(******************提示*******************)
bAnHaveLightWarn :=FALSE;
bCaHaveLightWarn :=FALSE;
FOR K1:=1 TO 50 DO 
      bAnHaveLightWarn:=bAnHaveLightWarn OR AnAlarm.arrLightWarn[K1];
	  bCaHaveLightWarn:=bCaHaveLightWarn OR CaAlarm.arrLightWarn[K1];
END_FOR
(***DDR负数报警***)
(***DDR负数报警***)
IF arrAxisCtrl[NameNo.CaAxisNo.DriverDDR].Status.fActPos<-1 THEN
	CaAlarm.arrFlowAlarm[30]:=TRUE;
END_IF
IF arrAxisCtrl[NameNo.AnAxisNo.DriverDDR].Status.fActPos<-1 THEN
	AnAlarm.arrFlowAlarm[30]:=TRUE;
END_IF

 IF   stSysState.bReset AND  AnAlarm.arrFlowAlarm[30] THEN
	    arrAxisCtrl[NameNo.AnAxisNo.DriverDDR].Cmd.fSetPos:=360;
		arrAxisCtrl[NameNo.AnAxisNo.DriverDDR].Cmd.bSetPos:=TRUE;
		AnAlarm.arrFlowAlarm[30]:=FALSE;
ELSIF  stSysState.bReset AND CaAlarm.arrFlowAlarm[30] THEN
	    arrAxisCtrl[NameNo.CaAxisNo.DriverDDR].Cmd.fSetPos:=360;
		arrAxisCtrl[NameNo.CaAxisNo.DriverDDR].Cmd.bSetPos:=TRUE;
		CaAlarm.arrFlowAlarm[30]:=FALSE;
 END_IF

 (******************报警复位*****************)
 FOR K3:=1 TO 98 DO 
	IF   stSysState.bReset AND  aAlarm[K3]AND NOT aAlarm[52] AND NOT aAlarm[53] AND NOT aAlarm[54]  THEN
			aAlarm[K3]:=FALSE;
	END_IF
END_FOR

(***气压不足报警***)
IF aAirAlarm_TON.Q THEN
	aAlarm[1]:=TRUE;
END_IF
YL_Q[1]:=aAlarm[1];//气压报警传给叠台；
(*
(*** R角废料清洁提示***)
IF  YL_GVL2[1]>=YL_GVL2[2] THEN//正极R角清废料报警；
	aAlarm[2]:=TRUE;
END_IF

IF  YL_GVL2[1]< 0 THEN//正极R角清废料计数错误；
	aAlarm[4]:=TRUE;
END_IF
///////////////////////////
IF    YL_GVL2[3] >=YL_GVL2[4] THEN//负极R角清废料报警；
	aAlarm[3]:=TRUE;
END_IF

IF  YL_GVL2[3] < 0 THEN//负极R角清废料计数错误；
	aAlarm[5]:=TRUE;
END_IF
/////////////////////////////
//复位
IF   stSysState.bReset AND  (aAlarm[2] OR  aAlarm[4] )THEN
		YL_GVL2[1]:=0;
		aAlarm[2]:=FALSE;
		aAlarm[4]:=FALSE;
END_IF

IF   stSysState.bReset AND  (aAlarm[3] OR  aAlarm[5] )THEN
		YL_GVL2[3]:=0;
		aAlarm[3]:=FALSE;
		aAlarm[5]:=FALSE;
END_IF
*)
(*** 除尘风机报警提示***)
aAlarm[6];//风机未启用报警；
IF NOT ProductPar.iModeEN.bFounctionClose[2] THEN
		IF NOT YL_I[1] OR NOT YL_I[3] OR NOT YL_I[5] OR NOT YL_I[7] THEN//2个5.5KW的吸片风机,2个除尘风机；
			aAlarm[6]:=TRUE;//风机未启用报警；
		END_IF
		IF  YL_I[2] OR YL_I[4] OR YL_I[6] OR YL_I[8]  THEN
			aAlarm[7]:=TRUE;// 风机故障报警；
		END_IF
END_IF
FanTon(IN:=NOT aAlarm[6]AND NOT FanTon.Q,PT:=T#1S,Q=>);
IF FanTon.Q THEN
	FanTonS:=FanTonS+1;
END_IF
IF FanTonS>=3600 THEN
	FanTonH:=FanTonH+1;
	FanTonS:=0;
END_IF
IF FanTonH_Set>=FanTonH THEN
	aAlarm[61]:=TRUE;;//风机寿命报警
END_IF



(*** 除尘毛刷气缸没有升起报警***)

IF stSysState.iMode=1 AND NOT 	arrCyCtrl[NameNo.AnCYNo.PoleBrushDustPush_U].Io.DIOFFSwitch THEN
				aAlarm[8]:=TRUE;//	正极上表面毛刷除尘升降气缸位置异常；
END_IF
IF stSysState.iMode=1 AND NOT	arrCyCtrl[NameNo.AnCYNo.PoleWindDustPush_U].Io.DIOFFSwitch THEN
				aAlarm[9]:=TRUE;//	正极上表面风刀除尘升降气缸位置异常;
END_IF
IF stSysState.iMode=1 AND NOT	arrCyCtrl[NameNo.AnCYNo.PoleBrushDustPush_D].Io.DIOFFSwitch THEN
				aAlarm[10]:=TRUE;//	正极下表面毛刷除尘升降气缸位置异常;
END_IF
IF stSysState.iMode=1 AND NOT	arrCyCtrl[NameNo.AnCYNo.PoleWindDustPush_D].Io.DIOFFSwitch THEN
				aAlarm[11]:=TRUE;//	//	正极下表面风刀除尘升降气缸位置异常;
END_IF
////////////////////////
IF stSysState.iMode=1 AND NOT 	arrCyCtrl[NameNo.CaCYNo.PoleBrushDustPush_U].Io.DIOFFSwitch THEN
				aAlarm[12]:=TRUE;//	负极上表面毛刷除尘升降气缸位置异常；
END_IF
IF stSysState.iMode=1 AND NOT	arrCyCtrl[NameNo.CaCYNo.PoleWindDustPush_U].Io.DIOFFSwitch THEN
				aAlarm[13]:=TRUE;//	负极上表面风刀除尘升降气缸位置异常;
END_IF
IF stSysState.iMode=1 AND NOT	arrCyCtrl[NameNo.CaCYNo.PoleBrushDustPush_D].Io.DIOFFSwitch THEN
				aAlarm[14]:=TRUE;//	负极下表面毛刷除尘升降气缸位置异常;
END_IF
IF stSysState.iMode=1 AND NOT	arrCyCtrl[NameNo.CaCYNo.PoleWindDustPush_D].Io.DIOFFSwitch THEN
				aAlarm[15]:=TRUE;//	负极下表面风刀除尘升降气缸位置异常;
END_IF

(*** 安全光栅报警***)
IF NOT AnSenser.biSafetyCurtain_M THEN
	aAlarm[16]:=TRUE;
END_IF
IF NOT AnSenser.biSafetyCurtain_C THEN
	aAlarm[17]:=TRUE;
END_IF		
	
IF NOT CaSenser.biSafetyCurtain_M THEN
	aAlarm[18]:=TRUE;
END_IF
IF NOT CaSenser.biSafetyCurtain_C THEN
	aAlarm[19]:=TRUE;
END_IF	
	
(***************风速仪报警**************)
(***************风速仪报警**************)

aTime[1](IN:=I107[8],PT:=T#20S,Q=>	);
aTime[2](IN:=I107[9],PT:=T#20S,Q=>	);
aTime[3](IN:=I107[10],PT:=T#20S,Q=>	);
aTime[4](IN:=I107[11],PT:=T#20S,Q=>	);
aTime[5](IN:=I107[12],PT:=T#20S,Q=>	);

aTime[6](IN:=I207[8],PT:=T#20S,Q=>	);
aTime[7](IN:=I207[9],PT:=T#20S,Q=>	);
aTime[8](IN:=I207[10],PT:=T#20S,Q=>	);
aTime[9](IN:=I207[11],PT:=T#20S,Q=>	);
aTime[10](IN:=I207[12],PT:=T#20S,Q=>);

IF NOT ProductPar.iModeEN.bFounctionClose[1] THEN//风速仪屏蔽
	IF aTime[1].Q THEN
		aAlarm[20]:=TRUE;
	END_IF
	IF aTime[2].Q THEN
		aAlarm[21]:=TRUE;
	END_IF
	IF aTime[3].Q THEN
		aAlarm[22]:=TRUE;
	END_IF
	IF aTime[4].Q THEN
		aAlarm[23]:=TRUE;
	END_IF
	IF aTime[5].Q THEN
		aAlarm[24]:=TRUE;
	END_IF
	IF aTime[6].Q THEN
		aAlarm[25]:=TRUE;
	END_IF
	IF aTime[7].Q THEN
		aAlarm[26]:=TRUE;
	END_IF
	IF aTime[8].Q THEN
		aAlarm[27]:=TRUE;
	END_IF
	IF aTime[9].Q THEN
		aAlarm[28]:=TRUE;
	END_IF
	IF aTime[10].Q THEN
		aAlarm[29]:=TRUE;
	END_IF
ELSE
	FOR i:=20 TO 29 DO
		aAlarm[i]:=FALSE;
	END_FOR	
END_IF
(******************毛刷感应报警********************)
FOR K4:=30 TO 47 DO 
     aAlarm[48]:=  aAlarm[K4];
END_FOR
(*
(***********摆杆电机扭矩值设置过小报警************)
IF iTargetTorque[1]>-20 THEN
	aAlarm[50]:=TRUE;//正极；
END_IF
IF iTargetTorque[2]>-20 THEN
	aAlarm[51]:=TRUE;//负极；
END_IF
*)
(****************模切清洁报警*********************)

CleanTrig(CLK:= (ProductPar.CleanTimeHMIHour1 = System.StTime.wHour AND ProductPar.CleanTimeHMIMin1 =System.stTime.wMinute)
OR (ProductPar.CleanTimeHMIHour2 = System.StTime.wHour AND ProductPar.CleanTimeHMIMin2 =System.stTime.wMinute)
OR (ProductPar.CleanTimeHMIHour3 = System.StTime.wHour AND ProductPar.CleanTimeHMIMin3 =System.stTime.wMinute)
OR (ProductPar.CleanTimeHMIHour4 = System.StTime.wHour AND ProductPar.CleanTimeHMIMin4 =System.stTime.wMinute));
IF CleanTrig.Q THEN
	aAlarm[52]:=TRUE;//请清洁机台
END_IF
(****************磁棒校验时间报警******************)
AnCibang(CLK:= (ProductPar.CibangTimeHMIHour1 = System.StTime.wHour AND ProductPar.CibangTimeHMIDay1 =System.stTime.wDay));
CaCibang(CLK:= (ProductPar.CibangTimeHMIHour2 = System.StTime.wHour AND ProductPar.CibangTimeHMIDay2 =System.stTime.wDay));
IF AnCibang.Q THEN
	aAlarm[53]:=TRUE;//正极磁棒校验时间报警
END_IF
IF CaCibang.Q THEN
	aAlarm[54]:=TRUE;//负极磁棒校验时间报警
END_IF
(****************模切毛刷清洁时间****************)
AnCleanBrush(CLK:= (ProductPar.BrushTimeHMIHour1 = System.StTime.wHour AND ProductPar.BrushTimeHMIDay1 =System.stTime.wDay));
CaCleanBrush(CLK:= (ProductPar.BrushTimeHMIHour2 = System.StTime.wHour AND ProductPar.BrushTimeHMIDay2 =System.stTime.wDay));
IF AnCleanBrush.Q THEN
	aAlarm[62]:=TRUE;//正极毛刷清洁时间报警
END_IF
IF CaCleanBrush.Q THEN
	aAlarm[63]:=TRUE;//负极毛刷清洁时间报警
END_IF

IF NOT  DTM_Mes1.bFuncEN[0] AND NOT ProductPar.iModeEN.bP2PartEN AND (DTM_Mes1.bFuncEN[1] OR DTM_Mes1.bFuncEN[2] OR DTM_Mes1.bFuncEN[3] OR
	        DTM_Mes1.bFuncEN[4] OR DTM_Mes1.bFuncEN[5] OR DTM_Mes1.bFuncEN[6] OR DTM_Mes1.bFuncEN[7] )  THEN
		 aAlarm[64]:=TRUE;//模切有功能屏蔽报警
END_IF		
			


 AnAlarm.arrFlowAlarm[9];
AnAlarm.arrFlowAlarm[10];
AnAlarm.arrFlowAlarm[11];
AnAlarm.arrFlowAlarm[12];
AnAlarm.arrFlowAlarm[13];
CaAlarm.arrFlowAlarm[9];
CaAlarm.arrFlowAlarm[10];
CaAlarm.arrFlowAlarm[11];
CaAlarm.arrFlowAlarm[12];
CaAlarm.arrFlowAlarm[13];
(*===============================================报警信息============================================================*)
(*****************报警汇总****************)////根据实际情况汇总
//正极报警汇总
arrError[1]:=bAnAxisHaveAlarm OR bAnCYHaveAlarm OR bAnTenHaveAlarm OR bAnCreatTableHaveAlarm OR bAnCamHaveAlarm OR bAnGearHaveAlarm OR bAnFlowHaveAlarm OR aAlarm[16] OR aAlarm[17] OR aAlarm[49]
		OR AnAlarm.arrFlowAlarm[9] OR AnAlarm.arrFlowAlarm[10] OR AnAlarm.arrFlowAlarm[11] OR AnAlarm.arrFlowAlarm[12] OR AnAlarm.arrFlowAlarm[13]
		OR CaAlarm.arrFlowAlarm[9] OR CaAlarm.arrFlowAlarm[10] OR CaAlarm.arrFlowAlarm[11] OR CaAlarm.arrFlowAlarm[12] OR CaAlarm.arrFlowAlarm[13] OR CuterCountAlarm[3];
//负极报警汇总
arrError[2]:=bCaAxisHaveAlarm OR bCaCYHaveAlarm OR bCaTenHaveAlarm OR bCaCreatTableHaveAlarm OR bCaCamHaveAlarm OR bCaGearHaveAlarm OR bCaFlowHaveAlarm OR aAlarm[18] OR aAlarm[19] OR aAlarm[49]
		OR AnAlarm.arrFlowAlarm[9] OR AnAlarm.arrFlowAlarm[10] OR AnAlarm.arrFlowAlarm[11] OR AnAlarm.arrFlowAlarm[12] OR AnAlarm.arrFlowAlarm[13]
		OR CaAlarm.arrFlowAlarm[9] OR CaAlarm.arrFlowAlarm[10] OR CaAlarm.arrFlowAlarm[11] OR CaAlarm.arrFlowAlarm[12] OR CaAlarm.arrFlowAlarm[13] OR CuterCountAlarm[6];
//提示
arrError[3]:=(ProductPar.iModeEN.iModeRun=0 AND (bAnHaveLightWarn OR bCaHaveLightWarn)) OR
				   (ProductPar.iModeEN.iModeRun=1 AND bAnHaveLightWarn) OR 
				   (ProductPar.iModeEN.iModeRun=2 AND bCaHaveLightWarn);

arrError[4];
arrError[5]:=CaAlarm.arrFlowAlarm[30] OR AnAlarm.arrFlowAlarm[30] OR aAlarm[1] OR aAlarm[2] OR aAlarm[3] OR aAlarm[4] OR aAlarm[5]  OR aAlarm[6] OR aAlarm[7] OR aAlarm[8] OR aAlarm[9]
					OR aAlarm[10] OR aAlarm[11] OR aAlarm[12] OR aAlarm[13] OR aAlarm[14] OR aAlarm[15]OR aAlarm[52]OR aAlarm[53]OR aAlarm[54] ;

stSysState.bErrorStop:=(ProductPar.iModeEN.iModeRun=0 AND (arrError[1] OR arrError[2])) OR
								   (ProductPar.iModeEN.iModeRun=1 AND arrError[1]) OR 
								   (ProductPar.iModeEN.iModeRun=2 AND arrError[2])OR arrError[5] OR aAlarm[64];
								   
								   
rDoorAlm[1](CLK:=(AnAlarm.arrFlowAlarm[9] OR AnAlarm.arrFlowAlarm[10] OR AnAlarm.arrFlowAlarm[11] OR AnAlarm.arrFlowAlarm[12] OR AnAlarm.arrFlowAlarm[13]) AND NOT
                            bAnAxisHaveAlarm AND NOT bAnCYHaveAlarm AND NOT bAnTenHaveAlarm AND NOT bAnCreatTableHaveAlarm AND NOT bAnCamHaveAlarm AND NOT
                           bAnGearHaveAlarm AND NOT bAnFlowHaveAlarm AND NOT aAlarm[16] AND NOT aAlarm[17] AND NOT aAlarm[49]  AND NOT CuterCountAlarm[3] );
rDoorAlm[2](CLK:=(CaAlarm.arrFlowAlarm[9] OR CaAlarm.arrFlowAlarm[10] OR CaAlarm.arrFlowAlarm[11] OR CaAlarm.arrFlowAlarm[12] OR CaAlarm.arrFlowAlarm[13]) AND NOT 
                            bCaAxisHaveAlarm AND NOT bCaCYHaveAlarm AND NOT bCaTenHaveAlarm AND NOT bCaCreatTableHaveAlarm AND NOT bCaCamHaveAlarm AND NOT 
                            bCaGearHaveAlarm AND NOT bCaFlowHaveAlarm AND NOT aAlarm[18] AND NOT aAlarm[19] AND NOT aAlarm[49]AND NOT CuterCountAlarm[6] );
IF 	rDoorAlm[1].Q OR bCaDoorALM THEN						
	bAnDoorALM:=TRUE;
END_IF			

IF 	rDoorAlm[1].Q THEN						
	bCaDoorALM:=TRUE;
END_IF		

IF NOT stSysState.bErrorStop AND bAnDoorALM THEN
	bAnDoorALM:=FALSE;
END_IF		
	
IF NOT stSysState.bErrorStop AND bCaDoorALM THEN
	bCaDoorALM:=FALSE;
END_IF				
(*==============报警复位=========================*)
//轴  气缸报警  红灯亮       蜂鸣器 0.5秒 频率 响 8 秒后停止    

IF stSysState.iMode=3 THEN
	stSysState.bReset:=stSysState.btnReset;
END_IF

(*****蜂鸣器*****)
rt100(CLK:=stSysState.bErrorStop, Q=> );
rt101(CLK:=arrError[3]  , Q=> );
IF rt100.Q THEN
	iErrorSetp:=100;//故障报警
END_IF

IF rt101.Q THEN
	iErrorSetp:=200;//警告报警
END_IF


tDelayBuzze(IN:= , PT:= , Q=> , ET=> );
CASE iErrorSetp   OF
100:
  tDelayBuzze.PT:=T#8S;
  tDelayBuzze.IN:=TRUE;
  iErrorSetp:=500;
200:
  tDelayBuzze.PT:=T#4S;
   tDelayBuzze.IN:=TRUE;
  iErrorSetp:=600;
500:
		stSysState.boBuzzer:= Pulse._250ms.Q;  //   (NOT bError1 AND NOT bError2) AND
		IF tDelayBuzze.Q  THEN
			iErrorSetp:=0;
			tDelayBuzze.IN:=FALSE;
			stSysState.boBuzzer:=FALSE;
		END_IF
600:
	IF stSysState.iMode=1 AND NOT stSysState.bErrorStop THEN
		stSysState.boRedLight:=Pulse._1s.Q;
	END_IF
		stSysState.boBuzzer:= Pulse._1s.Q;  //    (NOT bError1 AND NOT bError2) AND
		IF tDelayBuzze.Q  THEN
			iErrorSetp:=0;
			tDelayBuzze.IN:=FALSE;
			IF stSysState.iMode=1 AND NOT stSysState.bErrorStop THEN
				stSysState.boRedLight:=FALSE;
			END_IF
			stSysState.boBuzzer:=FALSE;
		END_IF

END_CASE


(*****三色灯控制*********)
//自动   绿
    RT200[1](CLK:=stSysState.iMode=1 AND NOT stSysState.bErrorStop , Q=> ); 
   IF RT200[1].Q THEN
	  bTurnOn:=TRUE;
      iLightSel:=3;
   END_IF       
//手动  黄
    RT200[2](CLK:=stSysState.iMode=3 AND NOT stSysState.bErrorStop , Q=> ); 
   IF RT200[2].Q THEN
	  bTurnOn:=TRUE;
      iLightSel:=2;
   END_IF 

//暂停   黄
    RT200[3](CLK:=stSysState.iMode=2 AND NOT stSysState.bErrorStop , Q=> ); 
   IF RT200[3].Q THEN
	  bTurnOn:=TRUE;
      iLightSel:=2;
   END_IF 
   
//暂停   红   //急停 OR 故障
    RT200[4](CLK:=stSysState.iMode=4  OR stSysState.bErrorStop  , Q=> ); 
   IF RT200[4].Q THEN
	  bTurnOn:=TRUE;
      iLightSel:=1;
   END_IF    
   
IF bTurnOn THEN
	CASE iLightSel OF 
	  1: //红灯
		stSysState.boGreenLight:=FALSE;
		stSysState.boRedLight:=TRUE;
		stSysState.boYellowLight:=FALSE;
	
	  2://黄灯
		stSysState.boGreenLight:=FALSE;
		stSysState.boRedLight:=FALSE;
		stSysState.boYellowLight:=TRUE;
	
	  3://绿灯
		stSysState.boGreenLight:=TRUE;
		stSysState.boRedLight:=FALSE;
		stSysState.boYellowLight:=FALSE;
	
	END_CASE
   bTurnOn:=FALSE;
END_IF
arrAxis[4].Status.Homed;
arrAxis[5].Status.Homed;
arrAxis[6].Status.Homed;
arrAxis[7].Status.Homed;
arrAxis[8].Status.Homed;
arrAxis[9].Status.Homed;
arrAxis[10].Status.Homed;
arrAxis[11].Status.Homed;
arrAxis[12].Status.Homed;
arrAxis[13].Status.Homed;
arrAxis[14].Status.Homed;
arrAxis[15].Status.Homed;
arrAxis[16].Status.Homed;
arrAxis[17].Status.Homed;
arrAxis[18].Status.Homed;
arrAxis[19].Status.Homed;
arrAxis[20].Status.Homed;
arrAxis[21].Status.Homed;
arrAxis[22].Status.Homed;
arrAxis[23].Status.Homed;
arrAxis[24].Status.Homed;
arrAxis[25].Status.Homed;
arrAxis[26].Status.Homed;
arrAxis[27].Status.Homed;
arrAxis[28].Status.Homed;
arrAxis[29].Status.Homed;
arrAxis[30].Status.Homed;
arrAxis[31].Status.Homed;
arrAxis[32].Status.Homed;
arrAxis[33].Status.Homed;
arrAxis[34].Status.Homed;
arrAxis[35].Status.Homed;
arrAxis[36].Status.Homed;
arrAxis[37].Status.Homed;
arrAxis[38].Status.Homed;
arrAxis[39].Status.Homed;
arrAxis[40].Status.Homed;
arrAxis[41].Status.Homed;
arrAxis[42].Status.Homed;
arrAxis[43].Status.Homed;
arrAxis[44].Status.Homed;
arrAxis[45].Status.Homed;
arrAxis[46].Status.Homed;
arrAxis[47].Status.Homed;
arrAxis[48].Status.Homed;
arrAxis[49].Status.Homed;
arrAxis[50].Status.Homed;
arrAxis[51].Status.Homed;
arrAxis[52].Status.Homed;
arrAxis[53].Status.Homed;
arrAxis[54].Status.Homed;
arrAxis[55].Status.Homed;
arrAxis[56].Status.Homed;
arrAxis[57].Status.Homed;
arrAxis[58].Status.Homed;
arrAxis[59].Status.Homed;
arrAxis[60].Status.Homed;
END_ACTION

ACTION Condition:
//按钮汇总
stSysState.btnAuto:=AnSys.btnAuto AND CaSys.btnAuto ;
stSysState.btnStart:=AnSys.btnStart OR CaSys.btnStart;
stSysState.btnStop:=AnSys.btnStop OR CaSys.btnStop;
stSysState.btnReset:=AnSys.btnReset OR CaSys.btnReset;
bEncloserEstop:=(NOT AnBtn.EncloserEstop[1] OR NOT AnBtn.EncloserEstop[2] OR NOT AnBtn.EncloserEstop[3] OR 
						  NOT CaBtn.EncloserEstop[1] OR NOT CaBtn.EncloserEstop[2] OR NOT CaBtn.EncloserEstop[3])AND test[1] ;
bBoxEstop:=NOT AnBtn.PoleBoxEStop OR NOT AnBtn.NGBoxEStop OR  NOT CaBtn.PoleBoxEStop OR NOT CaBtn.NGBoxEStop ;

stSysState.btnEstop:=(NOT AnSys.btnEstop OR NOT CaSys.btnEstop //面板急停
								OR bEncloserEstop//外罩急停
								(*OR bBoxEstop//按钮盒急停*)
								) ;//常闭
//面板按钮灯控制
bAnReady:=AnSys.bAutoCondition1 AND AnSys.Homed AND NOT AnSys.hmiDisCamAll;
bCaReady:=CaSys.bAutoCondition1 AND CaSys.Homed AND NOT CaSys.hmiDisCamAll;

AnSys.boStartLight:=stSysState.boGreenLight OR bAnReady AND Pulse._500ms.Q OR AnSys.btnStart;
CaSys.boStartLight:=stSysState.boGreenLight OR bCaReady AND Pulse._500ms.Q OR AnSys.btnStart;

AnSys.boStopLight:=AnSys.Stoping AND Pulse._250ms.Q OR AnSys.btnStop;
CaSys.boStopLight:=CaSys.Stoping AND Pulse._250ms.Q OR CaSys.btnStop;

AnSys.boResetLight:=stSysState.boRedLight AND Pulse._500ms.Q OR AnSys.btnReset;
CaSys.boResetLight:=stSysState.boRedLight AND Pulse._500ms.Q OR CaSys.btnReset;		
////////////////////////////////////////////设备状态//////////////////////
	IF stSysState.btnEstop THEN
		stSysState.iModehmi:=4;
	ELSIF NOT stSysState.btnEstop AND stSysState.bErrorStop THEN
		stSysState.iModehmi:=5;
	ELSIF NOT stSysState.btnEstop AND NOT stSysState.bErrorStop AND stSysState.FlgManua AND stSysState.iMode=3THEN
		stSysState.iModehmi:=3;
	ELSIF NOT stSysState.btnEstop AND NOT stSysState.bErrorStop AND ((NOT stSysState.FlgManua AND stSysState.FlgAuto AND stSysState.iMode=1) OR stSysState.iMode=1) THEN
		stSysState.iModehmi:=1;
	ELSIF NOT stSysState.btnEstop AND NOT stSysState.bErrorStop AND NOT stSysState.FlgManua AND stSysState.FlgAuto AND stSysState.iMode<>1 AND
		 	((ProductPar.iModeEN.iModeRun=0 AND bAnReady AND bCaReady) OR (ProductPar.iModeEN.iModeRun=1 AND bAnReady) OR (ProductPar.iModeEN.iModeRun=2 AND bCaReady))
			THEN	
		stSysState.iModehmi:=2;	
	ELSE
		stSysState.iModehmi:=6;	
	END_IF		
	P2Interaction.bP1Runing:=stSysState.iModehmi=1;
////////////////////////////////////////////主流程与分模块交互//////////////////////
(*
stSysState.bAutoCondition:=((AnSys.bAutoCondition1 AND AnSys.Homed AND NOT AnSys.hmiDisCamAll AND 
			CaSys.bAutoCondition1 AND CaSys.Homed AND NOT CaSys.hmiDisCamAll AND
			ProductPar.iModeEN.iModeRun=0) OR//正负同时启用
			(AnSys.bAutoCondition1 AND AnSys.Homed AND NOT AnSys.hmiDisCamAll AND
			ProductPar.iModeEN.iModeRun=1) OR//仅正极启用
			(CaSys.bAutoCondition1 AND CaSys.Homed AND NOT CaSys.hmiDisCamAll AND
			ProductPar.iModeEN.iModeRun=2))//仅负极启用
			AND NOT stSysState.bErrorStop;
*)
stSysState.bAutoCondition:=	(AnSys.bAutoCondition1 AND AnSys.Homed AND NOT AnSys.hmiDisCamAll AND CaSys.bAutoCondition1 AND CaSys.Homed AND NOT CaSys.hmiDisCamAll AND ProductPar.iModeEN.iModeRun=0 
	AND	( (ProductPar.AnPar.MQ.bWindSelect AND  Ansys.PolePieceNumberOK1)  OR ( NOT ProductPar.AnPar.MQ.bWindSelect AND  Ansys.PolePieceNumberOK2) )
	AND  ( ( ProductPar.CaPar.MQ.bWindSelect AND  Casys.PolePieceNumberOK1 ) OR (  NOT ProductPar.CaPar.MQ.bWindSelect AND  Casys.PolePieceNumberOK2 ) ) ) OR //正负同时启用

		(AnSys.bAutoCondition1 AND AnSys.Homed AND NOT AnSys.hmiDisCamAll AND ProductPar.iModeEN.iModeRun=1  AND
		 ( ( ProductPar.AnPar.MQ.bWindSelect AND  Ansys.PolePieceNumberOK1 ) OR (  NOT ProductPar.AnPar.MQ.bWindSelect AND  Ansys.PolePieceNumberOK2 ) )) OR//仅正极启用
	
		(CaSys.bAutoCondition1 AND CaSys.Homed AND NOT CaSys.hmiDisCamAll AND ProductPar.iModeEN.iModeRun=2 AND 
		  ( ( ProductPar.CaPar.MQ.bWindSelect AND  Casys.PolePieceNumberOK1 ) OR (  NOT ProductPar.CaPar.MQ.bWindSelect AND  Casys.PolePieceNumberOK2 )  ) )//仅负极启用
		  AND NOT stSysState.bErrorStop; 			
Ansys.bAutoTen:=stSysState.iMode=1 AND (ProductPar.iModeEN.iModeRun=0 OR ProductPar.iModeEN.iModeRun=1);
Casys.bAutoTen:=stSysState.iMode=1 AND (ProductPar.iModeEN.iModeRun=0 OR ProductPar.iModeEN.iModeRun=2);
Ansys.bAutoMain:=AnSys.bAutoCondition2 AND ((ProductPar.iModeEN.iModeRun=0 AND CaSys.bAutoCondition2) OR ProductPar.iModeEN.iModeRun=1);
Casys.bAutoMain:=CaSys.bAutoCondition2 AND ((ProductPar.iModeEN.iModeRun=0 AND AnSys.bAutoCondition2) OR ProductPar.iModeEN.iModeRun=2);

stSysState.bStopFinished:=(AnSys.bStopFinished AND CaSys.bStopFinished  AND ProductPar.iModeEN.iModeRun=0) OR//正负同时启用
			(AnSys.bStopFinished AND ProductPar.iModeEN.iModeRun=1) OR//仅正极启用
			(CaSys.bStopFinished AND ProductPar.iModeEN.iModeRun=2);//仅负极启用

///////////////////////////////////交互映射/////////////////////////////////////
//////////叠片TO模切//////////
//一号叠台正极
AnInter.M1Done:=D_Pro.bAn_M1Done;
AnInter.M1Safety:=D_Pro.bAn_M1Safety;
AnInter.iM1Ask:=D_Sys.iAn1Ask;
AnInter.M1LockReady:=D_Pro.bAn_M1LockReady;
AnInter.M1JumpReady:=D_Pro.bAn_M1JumpReady;
AnInter.M1PoleHave:=D_Pro.bAn_M1PoleHave;


//一号叠台负极
CaInter.M1Done:=D_Pro.bCa_M1Done;
CaInter.M1Safety:=D_Pro.bCa_M1Safety;
CaInter.iM1Ask:=D_Sys.iCa1Ask;
CaInter.M1LockReady:=D_Pro.bCa_M1LockReady;
CaInter.M1JumpReady:=D_Pro.bCa_M1JumpReady;
CaInter.M1PoleHave:=D_Pro.bCa_M1PoleHave;


//二号叠台正极
AnInter.M2Done:=D_Pro.bAn_M2Done;
AnInter.M2Safety:=D_Pro.bAn_M2Safety;
AnInter.iM2Ask:=D_Sys.iAn2Ask;
AnInter.M2LockReady:=D_Pro.bAn_M2LockReady;
AnInter.M2JumpReady:=D_Pro.bAn_M2JumpReady;
AnInter.M2PoleHave:=D_Pro.bAn_M2PoleHave;


//二号叠台负极
CaInter.M2Done:=D_Pro.bCa_M2Done;
CaInter.M2Safety:=D_Pro.bCa_M2Safety;
CaInter.iM2Ask:=D_Sys.iCa2Ask;
CaInter.M2LockReady:=D_Pro.bCa_M2LockReady;
CaInter.M2JumpReady:=D_Pro.bCa_M2JumpReady;
CaInter.M2PoleHave:=D_Pro.bCa_M2PoleHave;


//三号叠台正极
AnInter.M3Done:=D_Pro.bAn_M3Done;
AnInter.M3Safety:=D_Pro.bAn_M3Safety;
AnInter.iM3Ask:=D_Sys.iAn3Ask;
AnInter.M3LockReady:=D_Pro.bAn_M3LockReady;
AnInter.M3JumpReady:=D_Pro.bAn_M3JumpReady;
AnInter.M3PoleHave:=D_Pro.bAn_M3PoleHave;


//三号叠台负极
CaInter.M3Done:=D_Pro.bCa_M3Done;
CaInter.M3Safety:=D_Pro.bCa_M3Safety;
CaInter.iM3Ask:=D_Sys.iCa3Ask;
CaInter.M3LockReady:=D_Pro.bCa_M3LockReady;
CaInter.M3JumpReady:=D_Pro.bCa_M3JumpReady;
CaInter.M3PoleHave:=D_Pro.bCa_M3PoleHave;


//公共
P2Interaction.bP2ClearDo:=D_Sys.bP2ClearDo;
P2Interaction.bP2ClearDone:=D_Sys.bP2ClearDone;
P2Interaction.P2M1Enable:=D_Sys.bP2M1Enable;//叠台工位：1=屏蔽   模切工位：1=启用，故取反。
P2Interaction.P2M2Enable:=D_Sys.bP2M2Enable;//叠台工位：1=屏蔽   模切工位：1=启用，故取反。
P2Interaction.P2M3Enable:=D_Sys.bP2M3Enable;//叠台工位：1=屏蔽   模切工位：1=启用，故取反。
P2Interaction.bP2Estop:=D_Sys.bP2Estop;
P2Interaction.bP2Runing:=D_Sys.bP2Runing;
P2Interaction.bP2Start:=D_Sys.bP2Start;

///////////模切TO叠片/////////
//一号叠台正极
M_Pro.bAn_M1Allow:=AnInter.M1Allow;
M_Pro.bAn_M1Allow2:=AnInter.M1Allow2;
//一号叠台负极
M_Pro.bCa_M1Allow:=CaInter.M1Allow;
//M_Pro.bCa_M1Allow:=CaInter.M1Allow2;
//二号叠台正极
M_Pro.bAn_M2Allow:=AnInter.M2Allow;
//M_Pro.bAn_M2Allow2:=AnInter.M2Allow2;
//二号叠台负极
M_Pro.bCa_M2Allow:=CaInter.M2Allow;
//M_Pro.bCa_M2Allow:=CaInter.M2Allow2;
//三号叠台正极
M_Pro.bAn_M3Allow:=AnInter.M3Allow;
//M_Pro.bAn_M3Allow2:=AnInter.M3Allow2;
//三号叠台负极
M_Pro.bCa_M3Allow:=CaInter.M3Allow;
//M_Pro.bCa_M3Allow:=CaInter.M3Allow2;

(*20240404
///////////模切TO叠片/////////
//一号叠台正极
M_Pro.bAn_M1Allow:=AnInter.M1Allow;
//一号叠台负极
M_Pro.bCa_M1Allow:=CaInter.M1Allow;
//二号叠台正极
M_Pro.bAn_M2Allow:=AnInter.M2Allow;
//二号叠台负极
M_Pro.bCa_M2Allow:=CaInter.M2Allow;
//三号叠台正极
M_Pro.bAn_M3Allow:=AnInter.M3Allow;
//三号叠台负极
M_Pro.bCa_M3Allow:=CaInter.M3Allow;
20240404*)
//公共
M_Sys.bP1ClearDo:=P2Interaction.bP1ClearDo;
M_Sys.bP1ClearDone:=P2Interaction.bP1ClearDone;
M_Sys.bP1Estop:=P2Interaction.bP1Estop;
M_Sys.bP1Runing:=P2Interaction.bP1Runing;
M_Sys.bP1Start:=P2Interaction.bP1Start;
M_Sys.iCarryPoleMode:=ProductPar.iModeEN.iCarryPoleMode;
M_Sys.p1state:=stSysState.iModehmi;
IF test[2] THEN
	MEMSET(ADR(PoleData.AnIntervalData),0,SIZEOF(PoleData.AnIntervalData)); //  
	test[2]:=FALSE;
END_IF
IF test[3] THEN
	MEMSET(ADR(PoleData.CaIntervalData),0,SIZEOF(PoleData.CaIntervalData)); //  
	test[3]:=FALSE;
END_IF
IF test[4] THEN
	MEMSET(ADR(PoleData.AnTabData),0,SIZEOF(PoleData.AnTabData)); //  
	test[4]:=FALSE;
END_IF
IF test[5] THEN
	MEMSET(ADR(PoleData.CaTabData),0,SIZEOF(PoleData.CaTabData)); //  
	test[5]:=FALSE;
END_IF
//监控
PoleData.	AnBeltData[1].bHavePole;
PoleData.	AnBeltData[2].bHavePole;
PoleData.	AnBeltData[3].bHavePole;
PoleData.	AnBeltData[4].bHavePole;
PoleData.	AnBeltData[5].bHavePole;
PoleData.	AnBeltData[6].bHavePole;
PoleData.	AnBeltData[7].bHavePole;
PoleData.	AnBeltData[8].bHavePole;
PoleData.	AnBeltData[9].bHavePole;
PoleData.	AnBeltData[10].bHavePole;
PoleData.	AnBeltData[11].bHavePole;
PoleData.	AnBeltData[12].bHavePole;
PoleData.	AnBeltData[13].bHavePole;
PoleData.	AnBeltData[14].bHavePole;
PoleData.	AnBeltData[15].bHavePole;
PoleData.	AnBeltData[16].bHavePole;
PoleData.	AnBeltData[17].bHavePole;
PoleData.	AnBeltData[18].bHavePole;
PoleData.	AnBeltData[19].bHavePole;
PoleData.	AnBeltData[20].bHavePole;
PoleData.	AnBeltData[21].bHavePole;
PoleData.	AnBeltData[22].bHavePole;
PoleData.	AnBeltData[23].bHavePole;
PoleData.	AnBeltData[24].bHavePole;
PoleData.	AnBeltData[25].bHavePole;
PoleData.	AnBeltData[26].bHavePole;
PoleData.	AnBeltData[27].bHavePole;
PoleData.	AnBeltData[28].bHavePole;
PoleData.	AnBeltData[29].bHavePole;
PoleData.	AnBeltData[30].bHavePole;				
stSysState.hmiStart;					
bInitReset;
arrAxisCtrl[NameNo.AnVirAxisNo.VirMain].Status.fModuloActPos;
arrAxisCtrl[NameNo.AnVirAxisNo.VirDriver].Status.fActPos;
arrAxisCtrl[NameNo.AnVirAxisNo.VirBelt].Status.fActPos;
arrAxisCtrl[NameNo.AnAxisNo.Mould].Status.fModuloActPos;
arrAxisCtrl[NameNo.AnAxisNo.Cuter].Status.fModuloActPos;
arrAxisCtrl[NameNo.AnAxisNo.DriverDDR].Status.fActPos;
arrAxisCtrl[NameNo.AnAxisNo.CCDPressPush].Status.fModuloActPos;
//arrAxisCtrl[NameNo.AnAxisNo.NGPush2].Status.fModuloActPos;
arrAxisCtrl[NameNo.AnAxisNo.CuterBelt].Status.fActPos;
arrAxisCtrl[NameNo.AnAxisNo.NGPushReverseBelt].Status.fActPos;
arrAxisCtrl[NameNo.AnAxisNo.DedustBelt].Status.fActPos;
arrAxisCtrl[NameNo.AnAxisNo.DedustReverseBelt].Status.fActPos;
arrAxisCtrl[NameNo.AnAxisNo.SubBelt1].Status.fActPos;
arrAxisCtrl[NameNo.AnAxisNo.SubBelt2].Status.fActPos;
arrAxisCtrl[NameNo.AnAxisNo.SubBelt3].Status.fActPos;

arrAxisCtrl[NameNo.AnAxisNo.CuterBeltChange].Status.Homed;
arrAxisCtrl[NameNo.AnAxisNo.CuterBeltChange].cmd.bHome;

PoleData.	CaBeltData[1].bHavePole;
PoleData.	CaBeltData[2].bHavePole;
PoleData.	CaBeltData[3].bHavePole;
PoleData.	CaBeltData[4].bHavePole;
PoleData.	CaBeltData[5].bHavePole;
PoleData.	CaBeltData[6].bHavePole;
PoleData.	CaBeltData[7].bHavePole;
PoleData.	CaBeltData[8].bHavePole;
PoleData.	CaBeltData[9].bHavePole;
PoleData.	CaBeltData[10].bHavePole;
PoleData.	CaBeltData[11].bHavePole;
PoleData.	CaBeltData[12].bHavePole;
PoleData.	CaBeltData[13].bHavePole;
PoleData.	CaBeltData[14].bHavePole;
PoleData.	CaBeltData[15].bHavePole;
PoleData.	CaBeltData[16].bHavePole;
PoleData.	CaBeltData[17].bHavePole;
PoleData.	CaBeltData[18].bHavePole;
PoleData.	CaBeltData[19].bHavePole;
PoleData.	CaBeltData[20].bHavePole;
PoleData.	CaBeltData[21].bHavePole;
PoleData.	CaBeltData[22].bHavePole;
PoleData.	CaBeltData[23].bHavePole;
PoleData.	CaBeltData[24].bHavePole;
PoleData.	CaBeltData[25].bHavePole;
PoleData.	CaBeltData[26].bHavePole;
PoleData.	CaBeltData[27].bHavePole;
PoleData.	CaBeltData[28].bHavePole;
PoleData.	CaBeltData[29].bHavePole;
PoleData.	CaBeltData[30].bHavePole;	




//正极左卷料号OK
IF  (ProductPar.AnPar.MQ.bWindSelect AND arrCyCtrl[NameNo.AnCYNo.Inflation_L].Status.ONState 
 AND DT_To_MQ_MES.Mes_PcToPlc1 AND  LEN(DT_To_MQ_MES.PostiveCode1)>6  )  OR ProductPar.iModeEN.PartNumberOff THEN
	Ansys.PolePieceNumberOK1:=TRUE;
ELSE
	Ansys.PolePieceNumberOK1:=FALSE;
END_IF

//正极右卷料号OK
IF  (NOT ProductPar.AnPar.MQ.bWindSelect AND arrCyCtrl[NameNo.AnCYNo.Inflation_R].Status.ONState
  AND DT_To_MQ_MES.Mes_PcToPlc2 AND LEN(DT_To_MQ_MES.PostiveCode2)>6  )  OR ProductPar.iModeEN.PartNumberOff THEN
	Ansys.PolePieceNumberOK2:=TRUE;
ELSE
	Ansys.PolePieceNumberOK2:=FALSE;
END_IF

//当前使用左卷
IF ProductPar.AnPar.MQ.bWindSelect THEN
	IF Ansys.PolePieceNumberOK1 THEN
		PoleData.AnBeltData[1].Code:=DT_To_MQ_MES.PostiveCode1;
	ELSE
		PoleData.AnBeltData[1].Code:='';//当前卷物料码异常
	END_IF
ELSE//当前使用右卷
	IF Ansys.PolePieceNumberOK2 THEN
		PoleData.AnBeltData[1].Code:=DT_To_MQ_MES.PostiveCode2;
	ELSE
		PoleData.AnBeltData[1].Code:='';//当前卷物料码异常
	END_IF
END_IF

//正极右卷换左卷---正常换卷
Code_MES[1](CLK:=ProductPar.AnPar.MQ.bWindSelect , Q=> );//AND arrCyCtrl[NameNo.AnCYNo.Inflation_L].Status.ONState  AND  stAnUwindTen.bTensionOK 
IF Code_MES[1].Q THEN
	Ansys.PolePieceNumberOK2:=FALSE;//正极右卷料号OK
	MQ_To_DT_MES.Mes_PlcToPc1:=FALSE;//正极左卷换卷请求
	MQ_To_DT_MES.Mes_PlcToPc2:=TRUE;//正极右卷换卷请求触发
END_IF
//正极左卷换右卷---正常换卷
Code_MES[2](CLK:=NOT ProductPar.AnPar.MQ.bWindSelect  , Q=> );//AND arrCyCtrl[NameNo.AnCYNo.Inflation_R].Status.ONState  AND  stAnUwindTen.bTensionOK
IF Code_MES[2].Q THEN
	Ansys.PolePieceNumberOK1:=FALSE;//正极左卷料号OK
	MQ_To_DT_MES.Mes_PlcToPc1:=TRUE;//正极左卷换卷请求触发
	MQ_To_DT_MES.Mes_PlcToPc2:=FALSE;//正极右卷换卷请求
END_IF

//正极气涨轴切换换卷
Code_MES[3](CLK:=arrCyCtrl[NameNo.AnCYNo.Inflation_L].Io.DOStatus1, Q=> );//左卷
Code_MES[4](CLK:=arrCyCtrl[NameNo.AnCYNo.Inflation_R].Io.DOStatus1, Q=> );//右卷
IF Code_MES[3].Q THEN//左卷请求
	Ansys.PolePieceNumberOK1:=FALSE;//正极左卷料号OK
	MQ_To_DT_MES.Mes_PlcToPc1:=TRUE;//正极左卷换卷请求触发
	MQ_To_DT_MES.Mes_PlcToPc2:=FALSE;//正极右卷换卷请求
END_IF
IF Code_MES[4].Q THEN//右卷请求
	Ansys.PolePieceNumberOK2:=FALSE;//正极右卷料号OK
	MQ_To_DT_MES.Mes_PlcToPc1:=FALSE;//正极左卷换卷请求
	MQ_To_DT_MES.Mes_PlcToPc2:=TRUE;//正极右卷换卷请求触发
END_IF



//负极左卷料号OK
IF  (ProductPar.CaPar.MQ.bWindSelect AND arrCyCtrl[NameNo.CaCYNo.Inflation_L].Status.ONState 
 AND DT_To_MQ_MES.Mes_PcToPlc3 AND  LEN(DT_To_MQ_MES.NegativeCode1)>6  )  OR ProductPar.iModeEN.PartNumberOff THEN
	Casys.PolePieceNumberOK1:=TRUE;
ELSE
	Casys.PolePieceNumberOK1:=FALSE;
END_IF

//负极右卷料号OK
IF  (NOT ProductPar.CaPar.MQ.bWindSelect AND arrCyCtrl[NameNo.CaCYNo.Inflation_R].Status.ONState
  AND DT_To_MQ_MES.Mes_PcToPlc4 AND LEN(DT_To_MQ_MES.NegativeCode2)>6  )  OR ProductPar.iModeEN.PartNumberOff THEN
	Casys.PolePieceNumberOK2:=TRUE;
ELSE
	Casys.PolePieceNumberOK2:=FALSE;
END_IF

IF ProductPar.CaPar.MQ.bWindSelect THEN
	IF  Casys.PolePieceNumberOK1 THEN
		PoleData.CaBeltData[1].Code:=DT_To_MQ_MES.NegativeCode1;
	ELSE
		PoleData.CaBeltData[1].Code:='';//当前卷物料码异常
	END_IF
ELSE
	IF  Casys.PolePieceNumberOK2 THEN
		PoleData.CaBeltData[1].Code:=DT_To_MQ_MES.NegativeCode2;
	ELSE
		PoleData.CaBeltData[1].Code:='';//当前卷物料码异常
	END_IF
END_IF

//负极右卷换左卷---正常换卷
Code_MES[5](CLK:=ProductPar.CaPar.MQ.bWindSelect  , Q=> );//AND arrCyCtrl[NameNo.CaCYNo.Inflation_L].Status.ONState  AND  stCaUwindTen.bTensionOK
IF Code_MES[5].Q THEN
	Casys.PolePieceNumberOK2:=FALSE;//负极右卷料号OK
	MQ_To_DT_MES.Mes_PlcToPc3:=FALSE;//负极左卷换卷请求
	MQ_To_DT_MES.Mes_PlcToPc4:=TRUE;//负极右卷换卷请求触发
END_IF
//正极左卷换右卷---正常换卷
Code_MES[6](CLK:=NOT ProductPar.CaPar.MQ.bWindSelect  , Q=> );//AND arrCyCtrl[NameNo.CaCYNo.Inflation_R].Status.ONState  AND  stCaUwindTen.bTensionOK
IF Code_MES[6].Q THEN
	Casys.PolePieceNumberOK1:=FALSE;//负极左卷料号OK
	MQ_To_DT_MES.Mes_PlcToPc3:=TRUE;//负极左卷换卷请求触发
	MQ_To_DT_MES.Mes_PlcToPc4:=FALSE;//负极右卷换卷请求
END_IF


//负极气涨轴切换换卷
Code_MES[7](CLK:=arrCyCtrl[NameNo.CaCYNo.Inflation_L].Io.DOStatus1, Q=> );//左卷
Code_MES[8](CLK:=arrCyCtrl[NameNo.CaCYNo.Inflation_R].Io.DOStatus1, Q=> );//右卷
IF Code_MES[7].Q THEN//左卷请求
	Casys.PolePieceNumberOK1:=FALSE;//负极左卷料号OK
	MQ_To_DT_MES.Mes_PlcToPc3:=TRUE;//负极左卷换卷请求触发
	MQ_To_DT_MES.Mes_PlcToPc4:=FALSE;//负极右卷换卷请求
END_IF
IF Code_MES[8].Q THEN//右卷请求
	Casys.PolePieceNumberOK2:=FALSE;//负极右卷料号OK
	MQ_To_DT_MES.Mes_PlcToPc3:=FALSE;//负极左卷换卷请求
	MQ_To_DT_MES.Mes_PlcToPc4:=TRUE;//负极右卷换卷请求触发
END_IF



//条码校验未完成提示
IF ProductPar.AnPar.MQ.bWindSelect AND  NOT Ansys.PolePieceNumberOK1  AND NOT ProductPar.iModeEN.PartNumberOff THEN
	AnAlarm.arrLightWarn[41]:=TRUE;//正极左卷物料码校验未通过
ELSE
	AnAlarm.arrLightWarn[41]:=FALSE;//正极左卷物料码校验未通过
END_IF
IF NOT ProductPar.AnPar.MQ.bWindSelect AND NOT Ansys.PolePieceNumberOK2  AND NOT ProductPar.iModeEN.PartNumberOff THEN
	AnAlarm.arrLightWarn[42]:=TRUE;//正极右卷物料码校验未通过
ELSE
	AnAlarm.arrLightWarn[42]:=FALSE;//正极右卷物料码校验未通过
END_IF

IF ProductPar.CaPar.MQ.bWindSelect AND  NOT Casys.PolePieceNumberOK1  AND NOT ProductPar.iModeEN.PartNumberOff THEN
	CaAlarm.arrLightWarn[41]:=TRUE;//负极左卷物料码校验未通过
ELSE
	CaAlarm.arrLightWarn[41]:=FALSE;//负极左卷物料码校验未通过
END_IF
IF NOT  ProductPar.CaPar.MQ.bWindSelect AND NOT Casys.PolePieceNumberOK2  AND NOT ProductPar.iModeEN.PartNumberOff THEN
	CaAlarm.arrLightWarn[42]:=TRUE;//负极右卷物料码校验未通过
ELSE
	CaAlarm.arrLightWarn[42]:=FALSE;//负极右卷物料码校验未通过
END_IF


//触发信号清除
tCode_MES[1](IN:=MQ_To_DT_MES.Mes_PlcToPc1 , PT:=T#0.2S , Q=> , ET=> );
tCode_MES[2](IN:=MQ_To_DT_MES.Mes_PlcToPc2 , PT:=T#0.2S , Q=> , ET=> );
tCode_MES[3](IN:=MQ_To_DT_MES.Mes_PlcToPc3 , PT:=T#0.2S , Q=> , ET=> );
tCode_MES[4](IN:=MQ_To_DT_MES.Mes_PlcToPc4 , PT:=T#0.2S , Q=> , ET=> );
IF tCode_MES[1].Q THEN
	MQ_To_DT_MES.Mes_PlcToPc1:=FALSE;//正极左卷换卷请求触发
END_IF
IF tCode_MES[2].Q THEN
	MQ_To_DT_MES.Mes_PlcToPc2:=FALSE;//正极右卷换卷请求触发
END_IF
IF tCode_MES[3].Q THEN
	MQ_To_DT_MES.Mes_PlcToPc3:=FALSE;//负极左卷换卷请求触发
END_IF
IF tCode_MES[4].Q THEN
	MQ_To_DT_MES.Mes_PlcToPc4:=FALSE;//负极右卷换卷请求触发
END_IF


//料号相同检测
IF  NOT ProductPar.iModeEN.PartNumberOff  THEN
	IF DT_To_MQ_MES.PostiveCode1 =DT_To_MQ_MES.PostiveCode2 AND DT_To_MQ_MES.PostiveCode1<>''  THEN
		aAlarm[55]:=TRUE;;//正极左卷和正极右卷料号相同
	END_IF
	IF DT_To_MQ_MES.PostiveCode1 =DT_To_MQ_MES.NegativeCode1 AND DT_To_MQ_MES.PostiveCode1<>''  THEN
		aAlarm[56]:=TRUE;;//正极左卷和负极左卷料号相同
	END_IF
	IF DT_To_MQ_MES.PostiveCode1 =DT_To_MQ_MES.NegativeCode2 AND DT_To_MQ_MES.PostiveCode1<>''  THEN
		aAlarm[57]:=TRUE;;//正极左卷与负极右卷料号相同
	END_IF
	
	IF DT_To_MQ_MES.PostiveCode2 =DT_To_MQ_MES.NegativeCode1 AND DT_To_MQ_MES.PostiveCode2<>''  THEN
		aAlarm[58]:=TRUE;;//正极右卷和负极左卷料号相同
	END_IF
	IF DT_To_MQ_MES.PostiveCode2 =DT_To_MQ_MES.NegativeCode2 AND DT_To_MQ_MES.PostiveCode2<>'' THEN
		aAlarm[59]:=TRUE;;//正极右卷和负极右卷料号相同
	END_IF
	
	IF DT_To_MQ_MES.NegativeCode1= DT_To_MQ_MES.NegativeCode2 AND DT_To_MQ_MES.NegativeCode1<>'' THEN 
		aAlarm[60]:=TRUE;;//负极左卷和负极右卷料号相同
	END_IF
END_IF

IF YL_I[20] THEN//叠台一正极送片流水线安全点动条件 
		arrAxisCtrl[20].Cmd.JogN_Condition:=TRUE;
		arrAxisCtrl[20].Cmd.JogP_Condition:=TRUE;
ELSE
		arrAxisCtrl[20].Cmd.JogN_Condition:=FALSE;
		arrAxisCtrl[20].Cmd.JogP_Condition:=FALSE;	
END_IF
IF YL_I[21] THEN//叠台一负极送片流水线安全点动条件 
		arrAxisCtrl[44].Cmd.JogN_Condition:=TRUE;
		arrAxisCtrl[44].Cmd.JogP_Condition:=TRUE;
ELSE
		arrAxisCtrl[44].Cmd.JogN_Condition:=FALSE;
		arrAxisCtrl[44].Cmd.JogP_Condition:=FALSE;		
END_IF

IF YL_I[22] THEN//叠台二正极送片流水线安全点动条件 
		arrAxisCtrl[21].Cmd.JogN_Condition:=TRUE;
		arrAxisCtrl[21].Cmd.JogP_Condition:=TRUE;
ELSE
		arrAxisCtrl[21].Cmd.JogN_Condition:=FALSE;
		arrAxisCtrl[21].Cmd.JogP_Condition:=FALSE;	
END_IF
IF YL_I[23] THEN//叠台二负极送片流水线安全点动条件 
		arrAxisCtrl[45].Cmd.JogN_Condition:=TRUE;
		arrAxisCtrl[45].Cmd.JogP_Condition:=TRUE;
ELSE
		arrAxisCtrl[45].Cmd.JogN_Condition:=FALSE;
		arrAxisCtrl[45].Cmd.JogP_Condition:=FALSE;	
END_IF

IF YL_I[24] THEN//叠台三正极送片流水线安全点动条件 
		arrAxisCtrl[22].Cmd.JogN_Condition:=TRUE;
		arrAxisCtrl[22].Cmd.JogP_Condition:=TRUE;
ELSE
		arrAxisCtrl[22].Cmd.JogN_Condition:=FALSE;
		arrAxisCtrl[22].Cmd.JogP_Condition:=FALSE;	
END_IF
IF YL_I[25] THEN//叠台三负极送片流水线安全点动条件
		arrAxisCtrl[46].Cmd.JogN_Condition:=TRUE;
		arrAxisCtrl[46].Cmd.JogP_Condition:=TRUE;
ELSE
		arrAxisCtrl[46].Cmd.JogN_Condition:=FALSE;
		arrAxisCtrl[46].Cmd.JogP_Condition:=FALSE;	
END_IF
END_ACTION

ACTION CyBasic:

//气缸控制   刷新周期可以慢
FOR i:=1 TO MaxCy DO
    fbCy[i](bReset:=stSysState.bReset , CyCtrl:=arrCyCtrl[i] );
END_FOR
END_ACTION

ACTION EStop:
 FOR I1:=1 TO MaxAxes BY 1 DO
	arrAxisCtrl[I1].Cmd. bHome:=FALSE;
	arrAxisCtrl[I1].Cmd. bJog_Bw:=FALSE;	
	arrAxisCtrl[I1].Cmd. bJog_Fw:=FALSE;		
    arrAxisCtrl[I1].Cmd. bMoveAbs:=FALSE;		
    arrAxisCtrl[I1].Cmd. bMoveRel:=FALSE;	
    arrAxisCtrl[I1].Cmd. bMoveVelo:=FALSE;		
    arrAxisCtrl[I1].Cmd.bMoveModulo:=FALSE;	
    arrAxisCtrl[I1].Cmd. bSetPos:=FALSE;	    	
    arrAxisCtrl[I1].Cmd. iGoSetPos:=0;	  		
	arrAxisCtrl[NameNo.AnAxisNo.PoleTension].cmd.bEnable:=FALSE;
	arrAxisCtrl[NameNo.CaAxisNo.PoleTension].cmd.bEnable:=FALSE;
	arrAxisCtrl[I1].Cmd. bStop:=TRUE;		
  END_FOR;
 FOR I1:=1 TO MaxDust BY 1 DO
	arrDustMotor[I1].bRun_BW:=FALSE;
	arrDustMotor[I1].bRun_FW:=FALSE;	
  END_FOR
  
stAnUwindTen.bTenExecute:=FALSE;//正极放卷张力
stAnAuxDriverTen.bTenExecute:=FALSE;//正极张力辅助驱动			
		
stCaUwindTen.bTenExecute:=FALSE;//负极放卷张力						
stCaAuxDriverTen.bTenExecute:=FALSE;//负极张力辅助驱动
 



  stSysState.bInitDone:=FALSE;
  AnSys.bStopFinished:=FALSE; 
  CaSys.bStopFinished:=FALSE;
  stSysState.Stoping:=FALSE;
  AnSys.Homed:=FALSE;
  CaSys.Homed:=FALSE;


///////
	arrAxisCtrl[NameNo. AnVirAxisNo.VirMain].cmd.bEnable:=FALSE;
	arrAxisCtrl[NameNo. AnVirAxisNo.VirMain].cmd.bHalt:=FALSE;

	arrAxisCtrl[NameNo. CaVirAxisNo.VirMain].cmd.bEnable:=FALSE;
	arrAxisCtrl[NameNo. CaVirAxisNo.VirMain].cmd.bHalt:=FALSE;
END_ACTION

ACTION Init:

//整机初始化
//所有轴上使能，凸轮创建，时间轴跑速度

CASE iMainInitSetp OF
0:
    IF  NOT   stSysState.bInitDone THEN
         iMainInitSetp:=10;
    END_IF
10:
    FOR i:=1 TO MaxAxes DO 
		arrAxisCtrl[i].Cmd.bEnable:=TRUE;
		arrAxisCtrl[i].Cmd.bEnableFw:=TRUE;
		arrAxisCtrl[i].Cmd.bEnableBw:=TRUE;
	(*其他操作指令*)  
		arrAxisCtrl[i].Cmd.bHome:=FALSE;
		arrAxisCtrl[i].Cmd.bJog_Bw:=FALSE;
		arrAxisCtrl[i].Cmd.bHalt:=FALSE;
		arrAxisCtrl[i].Cmd.bJog_Fw:=FALSE;
		arrAxisCtrl[i].Cmd.bMoveAbs:=FALSE;
		arrAxisCtrl[i].Cmd.bMoveVelo:=FALSE;
		arrAxisCtrl[i].Cmd.bMoveRel:=FALSE;
		arrAxisCtrl[i].Cmd.bReset:=FALSE;
		arrAxisCtrl[i].Cmd.bStop:=FALSE;
		arrAxisCtrl[i].Cmd.bSetPos:=FALSE;
		
		//arrAxisCtrl[i].Cmd.JogN_Condition:=TRUE;
		//arrAxisCtrl[i].Cmd.JogP_Condition:=TRUE;
		arrAxisCtrl[i].Cmd.Home_Condition:=TRUE;
		
		
    END_FOR
    K1:=0;
    iMainInitSetp:=20;
20: //复位一次
   bInitReset:=TRUE;
   iMainInitSetp:=30;
30:
   K1:=K1+1;
   IF  K1>=10 THEN
        bInitReset:=FALSE;
        iMainInitSetp:=40;
   ELSE
     iMainInitSetp:=20;
   END_IF

40://正负极 Init
   AnSys.bInit:=TRUE;
   CaSys.bInit:=TRUE;
   AnSys.bInitDone:=FALSE;
   CaSys.bInitDone:=FALSE;
   iMainInitSetp:=50;
50:
   IF  AnSys.bInitDone AND CaSys.bInitDone THEN //  
        iMainInitSetp:=60;
	   // AnSys.bInitDone:=FALSE;
	   // CaSys.bInitDone:=FALSE;		
    END_IF

60: //复位一次
   bInitReset:=TRUE;
   iMainInitSetp:=70;
   
70: //Time 轴跑速度
  IF  arrAxis[NameNo.VirTimeWind].Status.ControlLoopClosed THEN
	  arrAxisPar[NameNo.VirTimeWind].fVelocity_of_Velo:=100;
	  arrAxisCtrl[NameNo.VirTimeWind].Cmd.bMoveVelo:=TRUE;
      bInitReset:=FALSE;
	  iMainInitSetp:=80;
  END_IF
 
80:
  IF arrAxis[NameNo.VirTimeWind].Status.ConstantVelocity THEN
        stSysState.bInitDone:=TRUE;
        iMainInitSetp:=0;
  END_IF

END_CASE
END_ACTION

ACTION MesCollect:
//xfp20240315 与MES交互优报表
ExcelRate_R(clk:=(DTM_Mes1.uOther[0]=1),Q=>);	//MES读取触发上升沿
IF ExcelRate_R.Q THEN	
	MTDWtStep:=10;
END_IF	

CASE MTDWtStep OF
	10:
		IF system.stTime.wHour >=8 AND system.stTime.wHour <20 THEN
			MTD_Mes1.rExcelRate[0]:=An_Production.NgPerHourDayCount[49];//正极极片尺寸NG总数量
			MTD_Mes1.rExcelRate[1]:=An_Production.NgPerHourDayCount[1];//正极极片长度不良
			MTD_Mes1.rExcelRate[2]:=An_Production.NgPerHourDayCount[2];//正极极片CIL宽度不良
			MTD_Mes1.rExcelRate[3]:=An_Production.NgPerHourDayCount[3];//正极极片宽度不良
			MTD_Mes1.rExcelRate[4]:=An_Production.NgPerHourDayCount[4];//正极极耳宽度不良
			MTD_Mes1.rExcelRate[5]:=An_Production.NgPerHourDayCount[5];//正极极耳高度不良
			MTD_Mes1.rExcelRate[6]:=An_Production.NgPerHourDayCount[6];//正极极耳侧边距不良
			MTD_Mes1.rExcelRate[7]:=An_Production.NgPerHourDayCount[7];//正极极耳面积不良
			MTD_Mes1.rExcelRate[8]:=An_Production.NgPerHourDayCount[8];//正极圆角深度不良
			MTD_Mes1.rExcelRate[9]:=An_Production.NgPerHourDayCount[9];//极耳边缘角度不良
			MTD_Mes1.rExcelRate[10]:=An_Production.NgPerHourDayCount[10];//正极圆角宽度不良
			MTD_Mes1.rExcelRate[11]:=An_Production.NgPerHourDayCount[11];//正极圆角轮廓不良
			MTD_Mes1.rExcelRate[12]:=An_Production.NgPerHourDayCount[12];//正极圆角面积不良
			MTD_Mes1.rExcelRate[13]:=An_Production.NgPerHourDayCount[13];//正极圆角余料不良
			MTD_Mes1.rExcelRate[14]:=An_Production.NgPerHourDayCount[14];//正极尺寸其它不良
			MTD_Mes1.rExcelRate[15]:=An_Production.NgPerHourDayCount[48];//正极片线扫NG总数量
			MTD_Mes1.rExcelRate[16]:=An_Production.NgPerHourDayCount[21];//正极片抓边失败
			MTD_Mes1.rExcelRate[17]:=An_Production.NgPerHourDayCount[22];//正极片直边不良
			MTD_Mes1.rExcelRate[18]:=An_Production.NgPerHourDayCount[23];//正极片极片缺失
			MTD_Mes1.rExcelRate[19]:=An_Production.NgPerHourDayCount[24];//正极片接带
			MTD_Mes1.rExcelRate[20]:=An_Production.NgPerHourDayCount[26];//正极片漏金属
			MTD_Mes1.rExcelRate[21]:=An_Production.NgPerHourDayCount[27];//正极片气泡
			MTD_Mes1.rExcelRate[22]:=An_Production.NgPerHourDayCount[28];//正极片暗条纹
			MTD_Mes1.rExcelRate[23]:=An_Production.NgPerHourDayCount[29];//正极片亮条纹
			MTD_Mes1.rExcelRate[24]:=An_Production.NgPerHourDayCount[30];//正极片破损
			MTD_Mes1.rExcelRate[25]:=An_Production.NgPerHourDayCount[32];//通信超时
			MTD_Mes1.rExcelRate[26]:=An_Production.NgPerHourDayCount[34];//正极片其它NG
			MTD_Mes1.rExcelRate[27]:=Ca_Production.NgPerHourDayCount[49];//负极极片尺寸NG总数量
			MTD_Mes1.rExcelRate[28]:=Ca_Production.NgPerHourDayCount[1];//负极极片长度不良
			MTD_Mes1.rExcelRate[29]:=Ca_Production.NgPerHourDayCount[3];//负极极片宽度不良
			MTD_Mes1.rExcelRate[30]:=Ca_Production.NgPerHourDayCount[4];//负极极耳宽度不良
			MTD_Mes1.rExcelRate[31]:=Ca_Production.NgPerHourDayCount[5];//负极极耳高度不良
			MTD_Mes1.rExcelRate[32]:=Ca_Production.NgPerHourDayCount[6];//负极极耳边距不良
			MTD_Mes1.rExcelRate[33]:=Ca_Production.NgPerHourDayCount[7];//负极极耳面积不良
			MTD_Mes1.rExcelRate[34]:=Ca_Production.NgPerHourDayCount[8];//负极圆角深度不良
			MTD_Mes1.rExcelRate[35]:=Ca_Production.NgPerHourDayCount[9];//极耳边缘角度不良
			MTD_Mes1.rExcelRate[36]:=Ca_Production.NgPerHourDayCount[10];//负极圆角宽度不良
			MTD_Mes1.rExcelRate[37]:=Ca_Production.NgPerHourDayCount[11];//负极圆角轮廓不良
			MTD_Mes1.rExcelRate[38]:=Ca_Production.NgPerHourDayCount[12];//负极圆角面积不良
			MTD_Mes1.rExcelRate[39]:=Ca_Production.NgPerHourDayCount[13];//负极圆角余料不良
			MTD_Mes1.rExcelRate[40]:=Ca_Production.NgPerHourDayCount[14];//负极尺寸其它不良
			MTD_Mes1.rExcelRate[41]:=Ca_Production.NgPerHourDayCount[48];//负极片线扫NG总数量
			MTD_Mes1.rExcelRate[42]:=Ca_Production.NgPerHourDayCount[21];//负极片抓边失败
			MTD_Mes1.rExcelRate[43]:=Ca_Production.NgPerHourDayCount[22];//负极片直边不良
			MTD_Mes1.rExcelRate[44]:=Ca_Production.NgPerHourDayCount[23];//负极片极片缺失
			MTD_Mes1.rExcelRate[45]:=Ca_Production.NgPerHourDayCount[24];//负极片接带
			MTD_Mes1.rExcelRate[46]:=Ca_Production.NgPerHourDayCount[26];//负极片漏金属
			MTD_Mes1.rExcelRate[47]:=Ca_Production.NgPerHourDayCount[27];//负极片气泡
			MTD_Mes1.rExcelRate[48]:=Ca_Production.NgPerHourDayCount[28];//负极片暗条纹
			MTD_Mes1.rExcelRate[49]:=Ca_Production.NgPerHourDayCount[29];//负极片亮条纹
			MTD_Mes1.rExcelRate[50]:=Ca_Production.NgPerHourDayCount[30];//负极片破损
			MTD_Mes1.rExcelRate[51]:=Ca_Production.NgPerHourDayCount[32];//通信超时
			MTD_Mes1.rExcelRate[52]:=Ca_Production.NgPerHourDayCount[34];//	负极片其它NG
			MTD_Mes1.rExcelRate[53]:=An_Production.NgPerHourDayCount[25];//	正极线扫黄标
			MTD_Mes1.rExcelRate[54]:=An_Production.NgPerHourDayCount[31];//	正极线扫碎屑
			MTD_Mes1.rExcelRate[55]:=An_Production.NgPerHourDayCount[33];//	正极线扫脱碳
			MTD_Mes1.rExcelRate[56]:=Ca_Production.NgPerHourDayCount[25];//	负极线扫黄标
			MTD_Mes1.rExcelRate[57]:=Ca_Production.NgPerHourDayCount[31];//	负极线扫碎屑
			MTD_Mes1.rExcelRate[58]:=Ca_Production.NgPerHourDayCount[33];//	负极线扫脱碳
			MTD_Mes1.uOther[0]:=2;	//plc数据写入完成
			MTDWtStep:=20;
		ELSIF system.stTime.wHour >=20 OR system.stTime.wHour<8 THEN	
			MTD_Mes1.rExcelRate[0]:=An_Production.NgPerHourNightCount[49];//正极极片尺寸NG总数量
			MTD_Mes1.rExcelRate[1]:=An_Production.NgPerHourNightCount[1];//正极极片长度不良
			MTD_Mes1.rExcelRate[2]:=An_Production.NgPerHourNightCount[2];//正极极片CIL宽度不良
			MTD_Mes1.rExcelRate[3]:=An_Production.NgPerHourNightCount[3];//正极极片宽度不良
			MTD_Mes1.rExcelRate[4]:=An_Production.NgPerHourNightCount[4];//正极极耳宽度不良
			MTD_Mes1.rExcelRate[5]:=An_Production.NgPerHourNightCount[5];//正极极耳高度不良
			MTD_Mes1.rExcelRate[6]:=An_Production.NgPerHourNightCount[6];//正极极耳侧边距不良
			MTD_Mes1.rExcelRate[7]:=An_Production.NgPerHourNightCount[7];//正极极耳面积不良
			MTD_Mes1.rExcelRate[8]:=An_Production.NgPerHourNightCount[8];//正极圆角深度不良
			MTD_Mes1.rExcelRate[9]:=An_Production.NgPerHourNightCount[9];//极耳边缘角度不良
			MTD_Mes1.rExcelRate[10]:=An_Production.NgPerHourNightCount[10];//正极圆角宽度不良
			MTD_Mes1.rExcelRate[11]:=An_Production.NgPerHourNightCount[11];//正极圆角轮廓不良
			MTD_Mes1.rExcelRate[12]:=An_Production.NgPerHourNightCount[12];//正极圆角面积不良
			MTD_Mes1.rExcelRate[13]:=An_Production.NgPerHourNightCount[13];//正极圆角余料不良
			MTD_Mes1.rExcelRate[14]:=An_Production.NgPerHourNightCount[14];//正极尺寸其它不良
			MTD_Mes1.rExcelRate[15]:=An_Production.NgPerHourNightCount[48];//正极片线扫NG总数量
			MTD_Mes1.rExcelRate[16]:=An_Production.NgPerHourNightCount[21];//正极片抓边失败
			MTD_Mes1.rExcelRate[17]:=An_Production.NgPerHourNightCount[22];//正极片直边不良
			MTD_Mes1.rExcelRate[18]:=An_Production.NgPerHourNightCount[23];//正极片极片缺失
			MTD_Mes1.rExcelRate[19]:=An_Production.NgPerHourNightCount[24];//正极片接带
			MTD_Mes1.rExcelRate[20]:=An_Production.NgPerHourNightCount[26];//正极片漏金属
			MTD_Mes1.rExcelRate[21]:=An_Production.NgPerHourNightCount[27];//正极片气泡
			MTD_Mes1.rExcelRate[22]:=An_Production.NgPerHourNightCount[28];//正极片亮条纹
			MTD_Mes1.rExcelRate[23]:=An_Production.NgPerHourNightCount[29];//正极片亮条纹
			MTD_Mes1.rExcelRate[24]:=An_Production.NgPerHourNightCount[30];//正极片破损
			MTD_Mes1.rExcelRate[25]:=An_Production.NgPerHourNightCount[32];//通信超时
			MTD_Mes1.rExcelRate[26]:=An_Production.NgPerHourNightCount[34];//正极片其它NG
			MTD_Mes1.rExcelRate[27]:=Ca_Production.NgPerHourNightCount[49];//负极极片尺寸NG总数量
			MTD_Mes1.rExcelRate[28]:=Ca_Production.NgPerHourNightCount[1];//负极极片长度不良
			MTD_Mes1.rExcelRate[29]:=Ca_Production.NgPerHourNightCount[3];//负极极片宽度不良
			MTD_Mes1.rExcelRate[30]:=Ca_Production.NgPerHourNightCount[4];//负极极耳宽度不良
			MTD_Mes1.rExcelRate[31]:=Ca_Production.NgPerHourNightCount[5];//负极极耳高度不良
			MTD_Mes1.rExcelRate[32]:=Ca_Production.NgPerHourNightCount[6];//负极极耳边距不良
			MTD_Mes1.rExcelRate[33]:=Ca_Production.NgPerHourNightCount[7];//负极极耳面积不良
			MTD_Mes1.rExcelRate[34]:=Ca_Production.NgPerHourNightCount[8];//负极圆角深度不良
			MTD_Mes1.rExcelRate[35]:=Ca_Production.NgPerHourNightCount[9];//极耳边缘角度不良
			MTD_Mes1.rExcelRate[36]:=Ca_Production.NgPerHourNightCount[10];//负极圆角宽度不良
			MTD_Mes1.rExcelRate[37]:=Ca_Production.NgPerHourNightCount[11];//负极圆角轮廓不良
			MTD_Mes1.rExcelRate[38]:=Ca_Production.NgPerHourNightCount[12];//负极圆角面积不良
			MTD_Mes1.rExcelRate[39]:=Ca_Production.NgPerHourNightCount[13];//负极圆角余料不良
			MTD_Mes1.rExcelRate[40]:=Ca_Production.NgPerHourNightCount[14];//负极尺寸其它不良
			MTD_Mes1.rExcelRate[41]:=Ca_Production.NgPerHourNightCount[48];//负极片线扫NG总数量
			MTD_Mes1.rExcelRate[42]:=Ca_Production.NgPerHourNightCount[21];//负极片抓边失败
			MTD_Mes1.rExcelRate[43]:=Ca_Production.NgPerHourNightCount[22];//负极片直边不良
			MTD_Mes1.rExcelRate[44]:=Ca_Production.NgPerHourNightCount[23];//负极片极片缺失
			MTD_Mes1.rExcelRate[45]:=Ca_Production.NgPerHourNightCount[24];//负极片接带
			MTD_Mes1.rExcelRate[46]:=Ca_Production.NgPerHourNightCount[26];//负极片漏金属
			MTD_Mes1.rExcelRate[47]:=Ca_Production.NgPerHourNightCount[27];//负极片气泡
			MTD_Mes1.rExcelRate[48]:=Ca_Production.NgPerHourNightCount[28];//负极片暗条纹
			MTD_Mes1.rExcelRate[49]:=Ca_Production.NgPerHourNightCount[29];//负极片亮条纹
			MTD_Mes1.rExcelRate[50]:=Ca_Production.NgPerHourNightCount[30];//负极片破损
			MTD_Mes1.rExcelRate[51]:=Ca_Production.NgPerHourNightCount[32];//通信超时
			MTD_Mes1.rExcelRate[52]:=Ca_Production.NgPerHourNightCount[34];//负极片其它NG
			MTD_Mes1.rExcelRate[53]:=An_Production.NgPerHourNightCount[25];//	正极线扫黄标
			MTD_Mes1.rExcelRate[54]:=An_Production.NgPerHourNightCount[31];//	正极线扫碎屑	
			MTD_Mes1.rExcelRate[55]:=An_Production.NgPerHourNightCount[33];//	正极线扫脱碳
			MTD_Mes1.rExcelRate[56]:=Ca_Production.NgPerHourNightCount[25];//	负极线扫黄标	
			MTD_Mes1.rExcelRate[57]:=Ca_Production.NgPerHourNightCount[31];//	负极线扫碎屑
			MTD_Mes1.rExcelRate[58]:=Ca_Production.NgPerHourNightCount[33];//	负极线扫脱碳
			MTD_Mes1.uOther[0]:=2;	//plc数据写入完成
			MTDWtStep:=20;
		END_IF			
	20:
		IF DTM_Mes1.uOther[0]=0 THEN
			MTD_Mes1.uOther[0]:=0;
			MTDWtStep:=0;
		END_IF
END_CASE
(*
//功能开关状态
        MTD_Mes1.bFuncEN[1]:=ProductPar.iModeEN.bCcdTcpEN;
		MTD_Mes1.bFuncEN[2]:=ProductPar.iModeEN.bLineScanCCDEN;
	    MTD_Mes1.bFuncEN[3]:=ProductPar.iModeEN.bChamferCCDEN;		
	    MTD_Mes1.bFuncEN[4]:=ProductPar.iModeEN.bCuterCCDEN;		
	    MTD_Mes1.bFuncEN[5]:=ProductPar.iModeEN.bSizeCCDEN;	
        MTD_Mes1.bFuncEN[6]:=ProductPar.iModeEN.PartNumberOff;
		MTD_Mes1.bFuncEN[7]:=ProductPar.iModeEN.bTabWidtNGoff;*)
		
//模具切刀计数		
		MTD_Mes1.uOther[1]:=ProductPar.AnPar.iCuterCount;
		MTD_Mes1.uOther[2]:=ProductPar.CaPar.iCuterCount;
		MTD_Mes1.uOther[3]:=ProductPar.AnPar.iMouldCount1;
		MTD_Mes1.uOther[4]:=ProductPar.CaPar.iMouldCount1;		
	    MTD_Mes1.uOther[5]:=ProductPar.AnPar.iCuterCountAlarm;
		MTD_Mes1.uOther[6]:=ProductPar.CaPar.iCuterCountAlarm;
		MTD_Mes1.uOther[7]:=ProductPar.AnPar.iMouldCountAlarm1;
		MTD_Mes1.uOther[8]:=ProductPar.CaPar.iMouldCountAlarm1;
		MTD_Mes1.bFuncEN[8]:=ProductPar.AnPar.iCuterclear;
		MTD_Mes1.bFuncEN[9]:=ProductPar.CaPar.iCuterclear;
		MTD_Mes1.bFuncEN[10]:=ProductPar.AnPar.iMouldclear1;
		MTD_Mes1.bFuncEN[11]:=ProductPar.CaPar.iMouldclear1;
END_ACTION

ACTION Motion_coe:

//nSlaveAddr :ARRAY[1..6] OF INT :=[1003,1008,1018,1019,1020,1021] ;     //EtherCAT支路驱动器ID



//////////////////////////////////////////////////////////////////////正极////////////////////////////////////////////////////////////////
(*
//正极模切缓存
//写入
FB_EcCoESdoWrite_AnSEPTATCache[1](
	sNetId:= '192.168.10.10.4.1', 
	nSlaveAddr:=1025,   //模切缓存
	nSubIndex:=0 , 
	nIndex:=16#2108 ,   //  平滑时间
	pSrcBuf:=ADR(SEPTATCache_fSmoothValue[1]),       //写入参数值 
	cbBufLen:=SIZEOF(SEPTATCache_fSmoothValue[1]),    
	bExecute:= SEPTATCache_bWriteCoeValue[1],    
	tTimeout:= T#3S, 
	bBusy=> , 
	bError=> , 
	nErrId=> );
//保存	
FB_EcCoESdoWrite_AnSEPTATCache[3](
	sNetId:= '192.168.10.10.4.1', 
	nSlaveAddr:=1025 ,   //模切缓存
	nSubIndex:=0 , 
	nIndex:=16#2108 ,   // 平滑时间
	pSrcBuf:=ADR(wSaveCoeCode),      //保存参数值
	cbBufLen:=SIZEOF(wSaveCoeCode),    
	bExecute:=SEPTATCache_SavePara[1],    
	tTimeout:= T#3S, 
	bBusy=> , 
	bError=> , 
	nErrId=> );	
	
	
//写入	
FB_EcCoESdoWrite_AnSEPTATCache[2](
	sNetId:='192.168.10.10.4.1', 
	nSlaveAddr:=1025 ,   //模切缓存
	nSubIndex:=0 , 
	nIndex:=16#2109 ,   // 平滑方式
	pSrcBuf:=ADR(SEPTATCache_fSmoothValue[2]),       //写入参数值 
	cbBufLen:=SIZEOF(SEPTATCache_fSmoothValue[2]),    
	bExecute:=SEPTATCache_bWriteCoeValue[2],    
	tTimeout:= T#3S, 
	bBusy=> , 
	bError=> , 
	nErrId=> );	
//保存
FB_EcCoESdoWrite_AnSEPTATCache[4](
	sNetId:= '192.168.10.10.4.1', 
	nSlaveAddr:=1025,   //模切缓存
	nSubIndex:=0 , 
	nIndex:=16#2109 ,   // 平滑方式
	pSrcBuf:=ADR(wSaveCoeCode),      //保存参数值
	cbBufLen:=SIZEOF(wSaveCoeCode),    
	bExecute:=SEPTATCache_SavePara[2],    
	tTimeout:= T#3S, 
	bBusy=> , 
	bError=> , 
	nErrId=> );	


	
	
	
	
//正极模切主驱
//写入
FB_EcCoESdoWrite_AnDriverDDR[1](
	sNetId:= '192.168.10.10.4.1', 
	nSlaveAddr:=1026 ,   //模切主驱
	nSubIndex:=0 , 
	nIndex:=16#2108 ,   //  平滑时间
	pSrcBuf:=ADR(DriverDDR_fSmoothValue[1]),       //写入参数值 
	cbBufLen:=SIZEOF(DriverDDR_fSmoothValue[1]),    
	bExecute:= DriverDDR_bWriteCoeValue[1],    
	tTimeout:= T#3S, 
	bBusy=> , 
	bError=> , 
	nErrId=> );
//保存	
FB_EcCoESdoWrite_AnDriverDDR[3](
	sNetId:= '192.168.10.10.4.1', 
	nSlaveAddr:=1026 ,   //模切主驱
	nSubIndex:=0 , 
	nIndex:=16#2108 ,   // 平滑时间
	pSrcBuf:=ADR(wSaveCoeCode),      //保存参数值
	cbBufLen:=SIZEOF(wSaveCoeCode),    
	bExecute:= DriverDDR_SavePara[1],    
	tTimeout:= T#3S, 
	bBusy=> , 
	bError=> , 
	nErrId=> );	
	
	
	
	
//写入	
FB_EcCoESdoWrite_AnDriverDDR[2](
	sNetId:='192.168.10.10.4.1', 
	nSlaveAddr:=1026 ,   //模切主驱
	nSubIndex:=0 , 
	nIndex:=16#2109 ,   // 平滑方式
	pSrcBuf:=ADR(DriverDDR_fSmoothValue[2]), 
	cbBufLen:=SIZEOF(DriverDDR_fSmoothValue[2]),    
	bExecute:= DriverDDR_bWriteCoeValue[2],    
	tTimeout:= T#3S, 
	bBusy=> , 
	bError=> , 
	nErrId=> );	
//保存
FB_EcCoESdoWrite_AnDriverDDR[4](
	sNetId:= '192.168.10.10.4.1', 
	nSlaveAddr:=1026 ,   //模切主驱
	nSubIndex:=0 , 
	nIndex:=16#2109 ,   // 平滑方式
	pSrcBuf:=ADR(wSaveCoeCode),  
	cbBufLen:=SIZEOF(wSaveCoeCode),    
	bExecute:= DriverDDR_SavePara[2],    
	tTimeout:= T#3S, 
	bBusy=> , 
	bError=> , 
	nErrId=> );	
			
	



	
	
	
	
	
	
	
	
	
	

//////////////////////////////////////////////////////////////////////负极////////////////////////////////////////////////////////////////////

//负极模切缓存
//写入
FB_EcCoESdoWrite_CaSEPTATCache[1](
	sNetId:= '192.168.10.10.4.1', 
	nSlaveAddr:=1041,   //模切缓存
	nSubIndex:=0 , 
	nIndex:=16#2108 ,   //  平滑时间
	pSrcBuf:=ADR(SEPTATCache_fSmoothValue[3]),       //写入参数值 
	cbBufLen:=SIZEOF(SEPTATCache_fSmoothValue[3]),    
	bExecute:= SEPTATCache_bWriteCoeValue[3],    
	tTimeout:= T#3S, 
	bBusy=> , 
	bError=> , 
	nErrId=> );
//保存	
FB_EcCoESdoWrite_CaSEPTATCache[3](
	sNetId:= '192.168.10.10.4.1', 
	nSlaveAddr:=1041 ,   //模切缓存
	nSubIndex:=0 , 
	nIndex:=16#2108 ,   // 平滑时间
	pSrcBuf:=ADR(wSaveCoeCode),      //保存参数值
	cbBufLen:=SIZEOF(wSaveCoeCode),    
	bExecute:= SEPTATCache_SavePara[3],    
	tTimeout:= T#3S, 
	bBusy=> , 
	bError=> , 
	nErrId=> );	
	
	
	
	
	
//写入	
FB_EcCoESdoWrite_CaSEPTATCache[2](
	sNetId:='192.168.10.10.4.1', 
	nSlaveAddr:=1041 ,   //模切缓存
	nSubIndex:=0 , 
	nIndex:=16#2109 ,   // 平滑方式
	pSrcBuf:=ADR(SEPTATCache_fSmoothValue[4]),       //写入参数值 
	cbBufLen:=SIZEOF(SEPTATCache_fSmoothValue[4]),    
	bExecute:= SEPTATCache_bWriteCoeValue[4],    
	tTimeout:= T#3S, 
	bBusy=> , 
	bError=> , 
	nErrId=> );
//保存	
FB_EcCoESdoWrite_CaSEPTATCache[4](
	sNetId:= '192.168.10.10.4.1', 
	nSlaveAddr:=1041,   //模切缓存
	nSubIndex:=0 , 
	nIndex:=16#2109 ,   // 平滑方式
	pSrcBuf:=ADR(wSaveCoeCode),      //保存参数值
	cbBufLen:=SIZEOF(wSaveCoeCode),    
	bExecute:= SEPTATCache_SavePara[4],    
	tTimeout:= T#3S, 
	bBusy=> , 
	bError=> , 
	nErrId=> );	


	
	
	
	

//负极模切主驱\
//写入
FB_EcCoESdoWrite_CaDriverDDR[1](
	sNetId:= '192.168.10.10.4.1', 
	nSlaveAddr:=1042 ,   //模切主驱
	nSubIndex:=0 , 
	nIndex:=16#2108 ,   //  平滑时间
	pSrcBuf:=ADR(DriverDDR_fSmoothValue[3]),       //写入参数值 
	cbBufLen:=SIZEOF(DriverDDR_fSmoothValue[3]),    
	bExecute:= DriverDDR_bWriteCoeValue[3],    
	tTimeout:= T#3S, 
	bBusy=> , 
	bError=> , 
	nErrId=> );
//保存	
FB_EcCoESdoWrite_CaDriverDDR[3](
	sNetId:= '192.168.10.10.4.1', 
	nSlaveAddr:=1042 ,   //模切主驱
	nSubIndex:=0 , 
	nIndex:=16#2108 ,   // 平滑时间
	pSrcBuf:=ADR(wSaveCoeCode),      //保存参数值
	cbBufLen:=SIZEOF(wSaveCoeCode),    
	bExecute:= DriverDDR_SavePara[3],    
	tTimeout:= T#3S, 
	bBusy=> , 
	bError=> , 
	nErrId=> );	
	
	
	
	
	
//写入	
FB_EcCoESdoWrite_CaDriverDDR[2](
	sNetId:='192.168.10.10.4.1', 
	nSlaveAddr:=1042 ,   //模切主驱
	nSubIndex:=0 , 
	nIndex:=16#2109 ,   // 平滑方式
	pSrcBuf:=ADR(DriverDDR_fSmoothValue[4]),       //写入参数值 
	cbBufLen:=SIZEOF(DriverDDR_fSmoothValue[4]),    
	bExecute:= DriverDDR_bWriteCoeValue[4],    
	tTimeout:= T#3S, 
	bBusy=> , 
	bError=> , 
	nErrId=> );	
//保存	
FB_EcCoESdoWrite_CaDriverDDR[4](
	sNetId:= '192.168.10.10.4.1', 
	nSlaveAddr:=1042 ,   //模切主驱
	nSubIndex:=0 , 
	nIndex:=16#2109 ,   // 平滑方式
	pSrcBuf:=ADR(wSaveCoeCode),      //保存参数值
	cbBufLen:=SIZEOF(wSaveCoeCode),    
	bExecute:= DriverDDR_SavePara[4],    
	tTimeout:= T#3S, 
	bBusy=> , 
	bError=> , 
	nErrId=> );	
	
	
	*)
END_ACTION

ACTION MotionBasic:


//
FOR i:=1 TO MaxAxes DO
IF i<>9 AND i<>33 AND i<>20 AND i<>21 AND i<>22 AND i<>44 AND i<>45 AND i<>46   THEN
  	arrAxisCtrl[i].Cmd.JogN_Condition:=NOT arrAxisCtrl[i].Io.biNegLimit;
	arrAxisCtrl[i].Cmd.JogP_Condition:=NOT arrAxisCtrl[i].Io.biPosLimit;
END_IF		
	csAxis[i](bReset:=stSysState.bReset , Axis:=arrAxis[i] , stAxisCtrl:=arrAxisCtrl[i] , stAxisPar:=arrAxisPar[i] );
	arrAxisPar[i].fHomeSlowSpeed:=arrAxisPar[i].fHomeFastSpeed/5;
END_FOR

FOR i:=1 TO MaxDust DO
  fbDustMotor[i](stSetpMotor:=arrDustMotor[i]);
END_FOR

FOR i:=1 TO NumOfDrives DO
  arrAxisCtrl[i].Status.bDrivesOP:=DrivesOP[i]=8;//(DrivesOP[i]=8 AND i<>3 AND i<>27) OR (DrivesOP[i]=10 AND (i=3 OR i=27));
END_FOR

fbAnSetp1Moter(stSetpMotor:=AnSetpMotor );//正极NG排杆电机
fbCaSetp1Moter(stSetpMotor:=CaSetpMotor );//负极NG排杆电机

IF ABS(iTargetTorque[1])>150 THEN
	iTargetTorque[1]:=0;
END_IF
IF ABS(iTargetTorque[2])>150 THEN
	iTargetTorque[2]:=0;
END_IF

//////////////张力摆杆超速后断开使能////////
IF (arrAxisCtrl[NameNo.AnAxisNo.PoleTension].Io.biNegLimit OR arrAxisCtrl[NameNo.AnAxisNo.PoleTension].Io.biPosLimit) AND arrAxisCtrl[NameNo.AnAxisNo.PoleTension].Status.fActVelo>500 THEN
	arrAxisCtrl[NameNo.AnAxisNo.PoleTension].Cmd.bEnable:=FALSE;
END_IF
IF (arrAxisCtrl[NameNo.CaAxisNo.PoleTension].Io.biNegLimit OR arrAxisCtrl[NameNo.CaAxisNo.PoleTension].Io.biPosLimit) AND arrAxisCtrl[NameNo.CaAxisNo.PoleTension].Status.fActVelo>500 THEN
	arrAxisCtrl[NameNo.CaAxisNo.PoleTension].Cmd.bEnable:=FALSE;
END_IF

//////////主轴参数放大////////
arrAxisPar[NameNo.AnVirAxisNo.VirMain].fMaxVel:=8000;
arrAxisPar[NameNo.AnVirAxisNo.VirMain].fMaxAccDec:=300000;
arrAxisPar[NameNo.AnVirAxisNo.VirMain].fConVelPercentage:=0.8;
arrAxisPar[NameNo.CaVirAxisNo.VirMain].fMaxVel:=8000;
arrAxisPar[NameNo.CaVirAxisNo.VirMain].fMaxAccDec:=300000;
arrAxisPar[NameNo.CaVirAxisNo.VirMain].fConVelPercentage:=0.8;
END_ACTION

ACTION MS_Alarm:
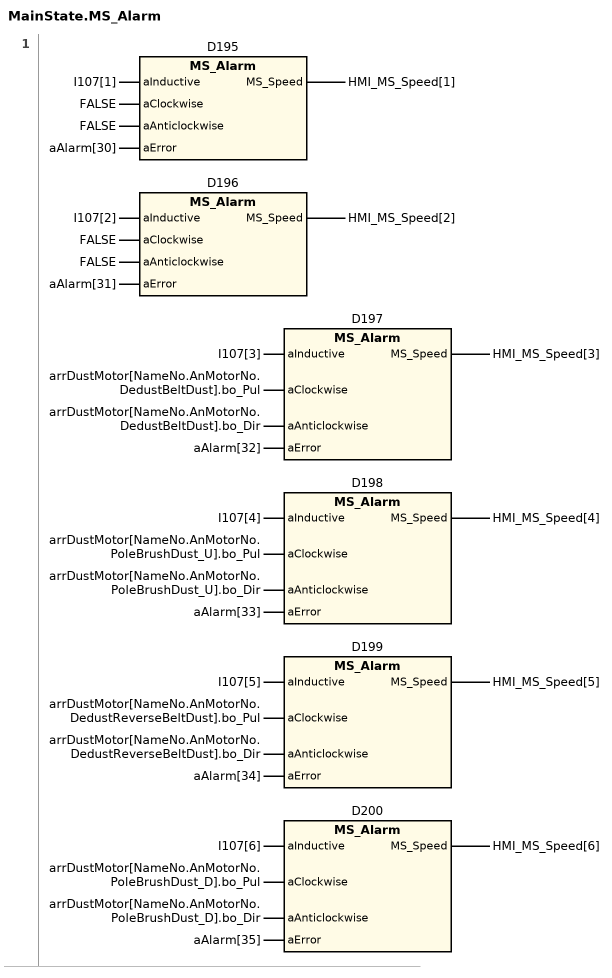
// NETWORK 1
D195(aInductive := I107[1], aClockwise := FALSE, aAnticlockwise := FALSE, aError := aAlarm[30]); // MS_Alarm
HMI_MS_Speed[1] := D195.MS_Speed;
D196(aInductive := I107[2], aClockwise := FALSE, aAnticlockwise := FALSE, aError := aAlarm[31]); // MS_Alarm
HMI_MS_Speed[2] := D196.MS_Speed;
D197(
    aInductive := I107[3],
    aClockwise := arrDustMotor[NameNo.AnMotorNo.DedustBeltDust].bo_Pul,
    aAnticlockwise := arrDustMotor[NameNo.AnMotorNo.DedustBeltDust].bo_Dir,
    aError := aAlarm[32]); // MS_Alarm
HMI_MS_Speed[3] := D197.MS_Speed;
D198(
    aInductive := I107[4],
    aClockwise := arrDustMotor[NameNo.AnMotorNo.PoleBrushDust_U].bo_Pul,
    aAnticlockwise := arrDustMotor[NameNo.AnMotorNo.PoleBrushDust_U].bo_Dir,
    aError := aAlarm[33]); // MS_Alarm
HMI_MS_Speed[4] := D198.MS_Speed;
D199(
    aInductive := I107[5],
    aClockwise := arrDustMotor[NameNo.AnMotorNo.DedustReverseBeltDust].bo_Pul,
    aAnticlockwise := arrDustMotor[NameNo.AnMotorNo.DedustReverseBeltDust].bo_Dir,
    aError := aAlarm[34]); // MS_Alarm
HMI_MS_Speed[5] := D199.MS_Speed;
D200(
    aInductive := I107[6],
    aClockwise := arrDustMotor[NameNo.AnMotorNo.PoleBrushDust_D].bo_Pul,
    aAnticlockwise := arrDustMotor[NameNo.AnMotorNo.PoleBrushDust_D].bo_Dir,
    aError := aAlarm[35]); // MS_Alarm
HMI_MS_Speed[6] := D200.MS_Speed;

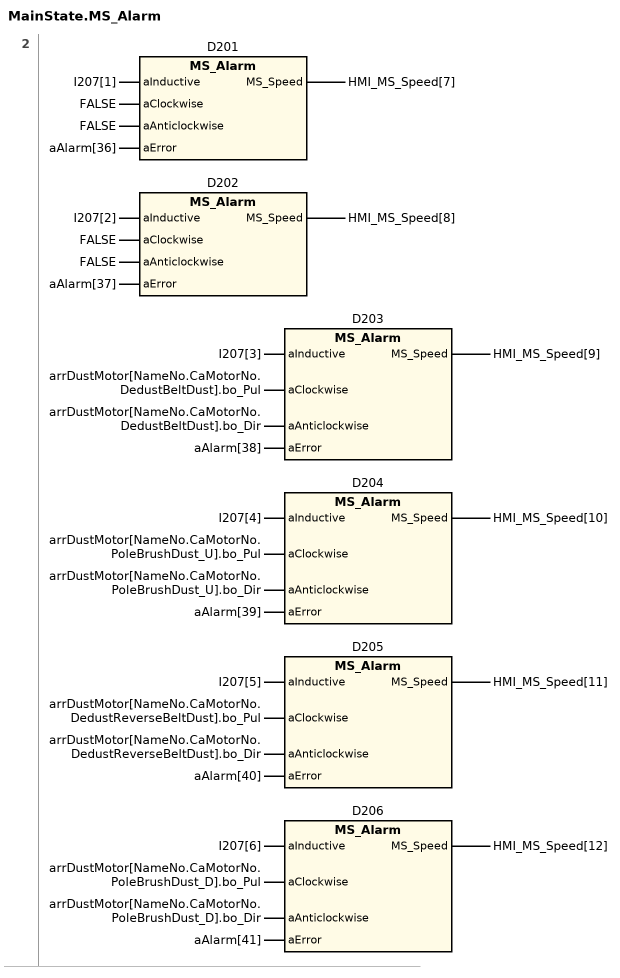
// NETWORK 2
D201(aInductive := I207[1], aClockwise := FALSE, aAnticlockwise := FALSE, aError := aAlarm[36]); // MS_Alarm
HMI_MS_Speed[7] := D201.MS_Speed;
D202(aInductive := I207[2], aClockwise := FALSE, aAnticlockwise := FALSE, aError := aAlarm[37]); // MS_Alarm
HMI_MS_Speed[8] := D202.MS_Speed;
D203(
    aInductive := I207[3],
    aClockwise := arrDustMotor[NameNo.CaMotorNo.DedustBeltDust].bo_Pul,
    aAnticlockwise := arrDustMotor[NameNo.CaMotorNo.DedustBeltDust].bo_Dir,
    aError := aAlarm[38]); // MS_Alarm
HMI_MS_Speed[9] := D203.MS_Speed;
D204(
    aInductive := I207[4],
    aClockwise := arrDustMotor[NameNo.CaMotorNo.PoleBrushDust_U].bo_Pul,
    aAnticlockwise := arrDustMotor[NameNo.CaMotorNo.PoleBrushDust_U].bo_Dir,
    aError := aAlarm[39]); // MS_Alarm
HMI_MS_Speed[10] := D204.MS_Speed;
D205(
    aInductive := I207[5],
    aClockwise := arrDustMotor[NameNo.CaMotorNo.DedustReverseBeltDust].bo_Pul,
    aAnticlockwise := arrDustMotor[NameNo.CaMotorNo.DedustReverseBeltDust].bo_Dir,
    aError := aAlarm[40]); // MS_Alarm
HMI_MS_Speed[11] := D205.MS_Speed;
D206(
    aInductive := I207[6],
    aClockwise := arrDustMotor[NameNo.CaMotorNo.PoleBrushDust_D].bo_Pul,
    aAnticlockwise := arrDustMotor[NameNo.CaMotorNo.PoleBrushDust_D].bo_Dir,
    aError := aAlarm[41]); // MS_Alarm
HMI_MS_Speed[12] := D206.MS_Speed;

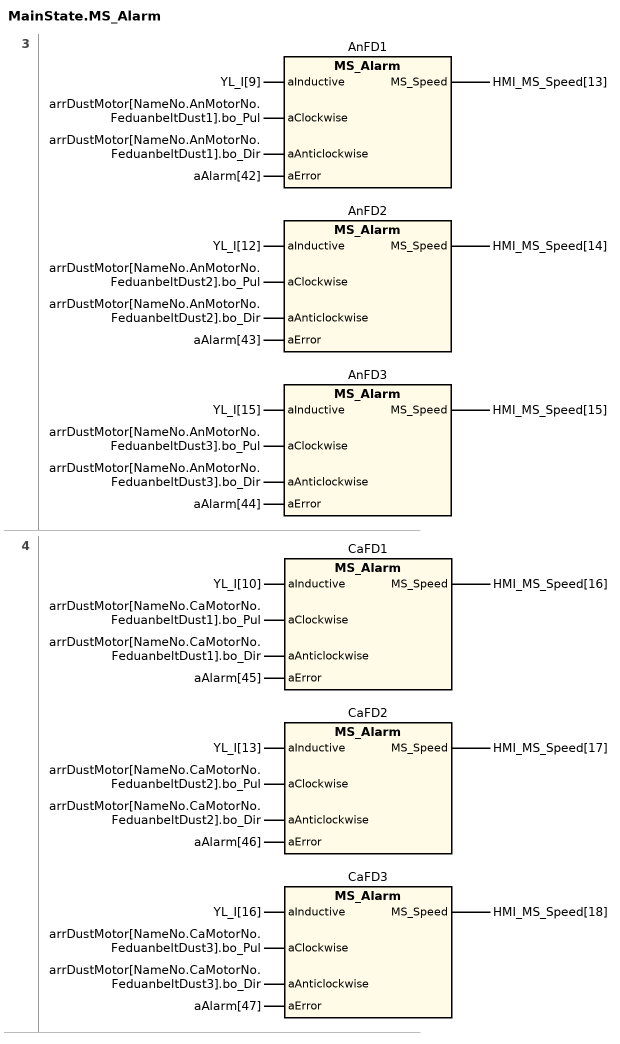
// NETWORK 3
AnFD1(
    aInductive := YL_I[9],
    aClockwise := arrDustMotor[NameNo.AnMotorNo.FeduanbeltDust1].bo_Pul,
    aAnticlockwise := arrDustMotor[NameNo.AnMotorNo.FeduanbeltDust1].bo_Dir,
    aError := aAlarm[42]); // MS_Alarm
HMI_MS_Speed[13] := AnFD1.MS_Speed;
AnFD2(
    aInductive := YL_I[12],
    aClockwise := arrDustMotor[NameNo.AnMotorNo.FeduanbeltDust2].bo_Pul,
    aAnticlockwise := arrDustMotor[NameNo.AnMotorNo.FeduanbeltDust2].bo_Dir,
    aError := aAlarm[43]); // MS_Alarm
HMI_MS_Speed[14] := AnFD2.MS_Speed;
AnFD3(
    aInductive := YL_I[15],
    aClockwise := arrDustMotor[NameNo.AnMotorNo.FeduanbeltDust3].bo_Pul,
    aAnticlockwise := arrDustMotor[NameNo.AnMotorNo.FeduanbeltDust3].bo_Dir,
    aError := aAlarm[44]); // MS_Alarm
HMI_MS_Speed[15] := AnFD3.MS_Speed;

// NETWORK 4
CaFD1(
    aInductive := YL_I[10],
    aClockwise := arrDustMotor[NameNo.CaMotorNo.FeduanbeltDust1].bo_Pul,
    aAnticlockwise := arrDustMotor[NameNo.CaMotorNo.FeduanbeltDust1].bo_Dir,
    aError := aAlarm[45]); // MS_Alarm
HMI_MS_Speed[16] := CaFD1.MS_Speed;
CaFD2(
    aInductive := YL_I[13],
    aClockwise := arrDustMotor[NameNo.CaMotorNo.FeduanbeltDust2].bo_Pul,
    aAnticlockwise := arrDustMotor[NameNo.CaMotorNo.FeduanbeltDust2].bo_Dir,
    aError := aAlarm[46]); // MS_Alarm
HMI_MS_Speed[17] := CaFD2.MS_Speed;
CaFD3(
    aInductive := YL_I[16],
    aClockwise := arrDustMotor[NameNo.CaMotorNo.FeduanbeltDust3].bo_Pul,
    aAnticlockwise := arrDustMotor[NameNo.CaMotorNo.FeduanbeltDust3].bo_Dir,
    aError := aAlarm[47]); // MS_Alarm
HMI_MS_Speed[18] := CaFD3.MS_Speed;
END_ACTION

ACTION Pusle:

/////////////////////////////////////////时钟脉冲////////////////////////////////////////////////////////////
//fbPulseCtrl1(PT_OFF:=T#2MS, PT_ON:=T#2MS, Q=>, RT=>);
fbPulseCtrl[1](PT_OFF:=T#2MS, PT_ON:=T#2MS,   );
fbPulseCtrl[2](PT_OFF:=T#4MS, PT_ON:=T#4MS,    );
fbPulseCtrl[3](PT_OFF:=T#10MS, PT_ON:=T#10MS,   );

fbPulseCtrl[4](PT_OFF:=T#50MS, PT_ON:=T#50MS,   );
fbPulseCtrl[5](PT_OFF:=T#3S, PT_ON:=T#3S,    );
fbPulseCtrl[6](PT_OFF:=T#5S, PT_ON:=T#5S,   );

fbPulseCtrl[8](PT_OFF:=T#250MS, PT_ON:=T#250MS,   );

fbPulseCtrl[9](PT_OFF:=T#2S, PT_ON:=T#200MS,   );
fbPulseCtrl[10](PT_OFF:=T#10S, PT_ON:=T#10S,   );
fbPulseCtrl[1].Q;
fbPulseCtrl[1].RT;
fbPulseCtrl[2].Q;
fbPulseCtrl[2].RT;
fbPulseCtrl[3].Q;
fbPulseCtrl[3].RT;
fbPulseCtrl[4].Q;
fbPulseCtrl[4].RT;
fbPulseCtrl[5].Q;
fbPulseCtrl[5].RT;
fbPulseCtrl[6].Q;
fbPulseCtrl[6].RT;

fbPulseCtrl[8].Q;
fbPulseCtrl[8].RT;
fbPulseCtrl[9].Q;
fbPulseCtrl[9].RT;
fbPulseCtrl[10].Q;
fbPulseCtrl[10].RT;
(*
IF bWaterOn AND ( bWaterOn2   OR    ABS( arrAxisCtrl[P1AxisNo.GMWind_U].Status.fActVelo)>=5 AND  ABS (arrAxisCtrl[P1AxisNo.GMWind_D].Status.fActVelo)>=5 )   THEN
  //P3EL2889S[3,5]:= fbPulseCtrl[9].Q;
   P1EL2889S[3,1]:= fbPulseCtrl[9].Q;
   P1EL2889S[3,2]:= fbPulseCtrl[9].Q;

   P2EL2889S[4,1]:=fbPulseCtrl[9].Q	;	
   P2EL2889S[4,2]:=fbPulseCtrl[9].Q;	

   P2EL2889S[4,3]:=fbPulseCtrl[9].Q	;	
   P2EL2889S[4,4]:=fbPulseCtrl[9].Q;	

ELSE
  //P3EL2889S[3,5]:= FALSE;
   P1EL2889S[3,1]:= FALSE;
   P1EL2889S[3,2]:= FALSE;
   P2EL2889S[4,1]:= FALSE	;	
   P2EL2889S[4,2]:= FALSE;	

   P2EL2889S[4,3]:=FALSE	;	
   P2EL2889S[4,4]:=FALSE;	
END_IF


//P1EL2889S[3,1]

*)
END_ACTION

ACTION RecBasic:
//纠偏控制
FOR i:=1 TO MaxRec DO
    fbRec[i]( RecCtrl:=arrRecCtrl[i] );
END_FOR
END_ACTION

END_PROGRAM

// ---- POUs/BasicFunction/Motion/MS_Alarm.TcPOU
FUNCTION_BLOCK MS_Alarm
VAR_INPUT
	aInductive:BOOL;//毛刷感应器；
	aClockwise:BOOL;//电机正转IO；
	aAnticlockwise:BOOL;//电机反转IO；
END_VAR
VAR_OUTPUT
	MS_Speed:REAL;//毛刷转速：r/min
END_VAR
VAR_IN_OUT//输入输出变量
	aError:BOOL;//毛刷未旋转感应报警；
END_VAR
VAR
	aTime1: TON;
	aTime2: TON;
	aTime3: TON;
	RunCount:INT;//毛刷感应器感应次数
	R_RunCount:R_TRIG;//毛刷感应器计数上升沿
	F_RunCount:F_TRIG;//毛刷感应器计数上升沿
	RunMark:BOOL;//毛刷运行标志
	RunCycle:INT;//毛刷运行周期
	RunCycleTime:REAL;//毛刷运行时间
	SpeedStep:INT;//毛刷速度计算运行步
	aInductiveMark:BOOL;
END_VAR

aTime1(IN:= aInductive AND (aClockwise OR aAnticlockwise),PT:=T#5S,Q=>	);
aTime2(IN:= NOT aInductive AND (aClockwise OR aAnticlockwise) ,PT:=T#5S,Q=>	);
IF aTime1.Q OR aTime2.Q THEN
	aError:=TRUE;
END_IF







//毛刷运行速度计算
	R_RunCount(CLK:= aInductive, Q=> );
	F_RunCount(CLK:= aInductive, Q=> );

	
	RunCount:=RunCount+1;//毛刷感应器感应次数	
	IF RunCount>=2000 THEN
		RunCount:=0;
	END_IF
	
	
	
	IF R_RunCount.Q THEN
		RunMark:=TRUE;//毛刷运行标志
		RunCycle:=RunCycle+1  ;//毛刷感应器感应次数	
	END_IF
	
	IF RunMark  THEN
		MS_Speed:=345+ RunCount/25+RunCycle;//毛刷运行周期
	END_IF
	
	
	IF RunCount=14 OR ((RunCount<13) AND NOT aClockwise AND NOT aAnticlockwise ) THEN
		RunCycleTime:=0;
		RunCount:=0;//毛刷感应器感应次数
		RunCycle:=0;//毛刷运行周期	
		RunMark:=FALSE;//毛刷运行标志
	END_IF











(*
//毛刷运行速度计算
	R_RunCount(CLK:= aInductive, Q=> );
	F_RunCount(CLK:= aInductive, Q=> );

	IF R_RunCount.Q THEN
		RunMark:=TRUE;//毛刷运行标志
		RunCount:=RunCount+1;//毛刷感应器感应次数	
	END_IF
	
	IF RunMark AND RunCount<13 THEN
		RunCycle:=RunCycle+1;//毛刷运行周期
	END_IF
	
	//RunCycleTime:=(RunCycle*2);//毛刷运行时间(S)
	
	IF RunCount=13 THEN
		RunCycleTime:=(RunCycle*2);//毛刷运行时间(S)
	END_IF
	IF RunCycleTime<>0 AND RunCount=13 THEN
		MS_Speed:=1000*((3/RunCycleTime)*60);//毛刷转速：r/min//1.17*
	END_IF
	IF RunCount=14 OR ((RunCount<13) AND NOT aClockwise AND NOT aAnticlockwise ) THEN
		RunCycleTime:=0;
		RunCount:=0;//毛刷感应器感应次数
		RunCycle:=0;//毛刷运行周期	
		RunMark:=FALSE;//毛刷运行标志
	END_IF
*)

END_FUNCTION_BLOCK

// ---- POUs/BasicFunction/Basic/05_Actuators/FB_CylinderV2.TcPOU
FUNCTION_BLOCK FB_CylinderV2
VAR_INPUT
	bReset	:	BOOL	;	
END_VAR

VAR_IN_OUT
  CyCtrl: ST_CyCtrl;
END_VAR


VAR
	rON	:	R_TRIG	;
	rOFF	:	R_TRIG	;
	rFree	:	R_TRIG	;
	Delay2	:	TON	;
	Delay3	:	TON	;
	RS1	:	RS	;
	RS2	:	RS	;
	Delay4	:	TON	;
	Delay5	:	TON	;
	rError1	:	R_TRIG	;
	fError2	:	F_TRIG	;
	fError1	:	F_TRIG	;
	rError2	:	R_TRIG	;
	DelayOnSwitch	:	TON	;
	DelayOffSwitch	:	TON	;
	M1	:	BOOL	;



END_VAR


rON(CLK:=CyCtrl.Cmd.bON );   
rOFF(CLK:=CyCtrl.Cmd.bOFF  );
rFree(CLK:=CyCtrl.Cmd.bFree  );

IF rON.Q THEN 
	CyCtrl.Cmd.bOFF:=FALSE;
    CyCtrl.Cmd.bFree :=FALSE;
END_IF;
IF rOFF.Q THEN 
	CyCtrl.Cmd.bON:=FALSE;
    CyCtrl.Cmd.bFree :=FALSE;
END_IF;
IF rFree.Q THEN 
	CyCtrl.Cmd.bON:=FALSE;
	CyCtrl.Cmd.bOFF:=FALSE;
END_IF;


IF   CyCtrl.Cmd.iType=1 OR CyCtrl.Cmd.iType=3   THEN  // 双
		IF   rON.Q THEN
				RS1.SET:=TRUE;
		        RS1.RESET1:=FALSE;
				RS2.SET:=FALSE;
		        RS2.RESET1:=TRUE;			
		END_IF;
		IF   rOFF.Q THEN
				RS2.SET:=TRUE;
		        RS2.RESET1:=FALSE;
				RS1.SET:=FALSE;
		       RS1.RESET1:=TRUE;		   
		END_IF;
END_IF;	

IF   CyCtrl.Cmd.iType=2  OR  CyCtrl.Cmd.iType=4   THEN  //   单
		IF   rON.Q THEN
				RS1.SET:=TRUE;
		       RS1.RESET1:=FALSE;
		END_IF;
		IF   rOFF.Q THEN
				RS1.SET:=FALSE;
		       RS1.RESET1:=TRUE;
		END_IF;
   
   	 RS2.SET:=FALSE;
	 RS2.RESET1:=TRUE;	  
END_IF;
  
IF  CyCtrl.Cmd.iType>=1 AND   CyCtrl.Cmd.iType<=3 THEN  //泄压
 	 IF   rFree.Q THEN
		RS1.SET:=FALSE;
		RS1.RESET1:=TRUE;		
		RS2.SET:=FALSE;
		RS2.RESET1:=TRUE;
   END_IF
END_IF

IF  CyCtrl.Cmd.iType=1 OR  CyCtrl.Cmd.iType=2 THEN
     CyCtrl.Status.ONState:=CyCtrl.Io.DIOnSwitch;
      CyCtrl.Status.OFFState:=CyCtrl.Io.DIOFFSwitch;
END_IF
IF  CyCtrl.Cmd.iType=4  THEN  
     CyCtrl.Status.ONState:=  CyCtrl.Io.DOStatus1;
      CyCtrl.Status.OFFState:=NOT CyCtrl.Io.DOStatus1;
END_IF
IF  CyCtrl.Cmd.iType=3  THEN  
     CyCtrl.Status.ONState:=CyCtrl.Io.DOStatus1;
      CyCtrl.Status.OFFState:=CyCtrl.Io.DOStatus2;
END_IF

(*
//仿真用
DelayOnSwitch(IN:=DOStatus1 , PT:=T#2000MS  );  //仿真用
DelayOffSwitch(IN:=DOStatus2 , PT:=T#2000MS  );

ONState:=DelayOnSwitch.Q;
OFFState:=DelayOffSwitch.Q;
   *)
RS1( Q1=>CyCtrl.Io.DOStatus1 );
RS2( Q1=>CyCtrl.Io.DOStatus2 );
///////////////////////////////////////
IF  CyCtrl.Cmd.iType=2 OR  CyCtrl.Cmd.iType=4  THEN  //   单控 T#100MS
	Delay4(IN:=(RS1.SET      AND  NOT  CyCtrl.Status.ONState) , PT:=INT_TO_TIME(CyCtrl.Cmd.ErrorTime)*1000  );//ON 到位报警
	Delay5(IN:=(RS1.RESET1 AND NOT  CyCtrl.Status.OFFState ) , PT:= INT_TO_TIME(CyCtrl.Cmd.ErrorTime)*1000  );//OFF 到位报警
	;
ELSIF  CyCtrl.Cmd.iType=1  OR  CyCtrl.Cmd.iType=3  THEN
	Delay4(IN:=(RS1.SET      AND  NOT  CyCtrl.Status.ONState) ,   PT:= INT_TO_TIME(CyCtrl.Cmd.ErrorTime)*1000     );//ON 到位报警
	Delay5(IN:=(RS2.SET      AND  NOT  CyCtrl.Status.OFFState ) , PT:=INT_TO_TIME(CyCtrl.Cmd.ErrorTime)*1000      );//OFF 到位报警 MULTIME(In1:=T#100MS, In2:=ErrorTime) 
	;
END_IF;
	


CyCtrl.Status.Error1:=Delay4.Q;
CyCtrl.Status.Error2:=Delay5.Q;





(*
rError1(CLK:=Delay4.Q  );  
rError2(CLK:=Delay5.Q  );  

IF rError1.Q THEN    
	CyCtrl.Status.Error1:=TRUE;
END_IF;

IF rError2.Q THEN    
	CyCtrl.Status.Error2:=TRUE;
END_IF;


IF bReset AND (  CyCtrl.Status.Error1 OR CyCtrl.Status.Error2 )THEN
	CyCtrl.Status.Error1:=FALSE;
	CyCtrl.Status.Error2:=FALSE;
END_IF;
*)

END_FUNCTION_BLOCK

// ---- POUs/BasicFunction/Motion/CS_DustMoter.TcPOU
FUNCTION_BLOCK CS_DustMoter
VAR_INPUT
END_VAR
VAR_OUTPUT
END_VAR
VAR
END_VAR

VAR_IN_OUT
stSetpMotor:ST_DustMotor;
END_VAR
	

VAR
R_trig20:R_TRIG;
R_trig21:R_TRIG;
F_trig23:F_TRIG;
F_trig22:F_TRIG;
END_VAR

(*********************毛刷步进电机控制*****************************)
//步进点动
stSetpMotor.bo_Pul:=stSetpMotor.bJog_FW OR stSetpMotor.bJog_BW ;   //步进点动正转
stSetpMotor.bo_Dir:=stSetpMotor.bJog_BW ; //步进点动反转   

R_trig20(CLK:=stSetpMotor.bRun_FW , Q=> );
R_trig21(CLK:=stSetpMotor.bRun_BW , Q=> );
F_trig22(CLK:=stSetpMotor.bRun_FW , Q=> );
F_trig23(CLK:=stSetpMotor.bRun_BW , Q=> );
IF R_trig20.Q THEN
   stSetpMotor.bJog_FW:=TRUE;
   stSetpMotor.bJog_BW:=FALSE;
END_IF
IF R_trig21.Q THEN
   stSetpMotor.bJog_FW:=FALSE;
   stSetpMotor.bJog_BW:=TRUE;
END_IF
IF F_trig22.Q OR F_trig23.Q THEN
   stSetpMotor.bJog_FW:=FALSE;
   stSetpMotor.bJog_BW:=FALSE;
END_IF

END_FUNCTION_BLOCK

// ---- POUs/BasicFunction/MES/CS_CodeTcp.TcPOU
FUNCTION_BLOCK PUBLIC CS_CodeTcp
VAR_INPUT
END_VAR
VAR_OUTPUT
END_VAR
VAR_IN_OUT
	
   iCode2:ICode;

END_VAR


VAR
	
	fbTcpCon:FB_SocketConnect;
	fbTcpSend:FB_SocketSend;
//	fbTcpSend2:FB_SocketSend;
	fbTcpRec:FB_SocketReceive;
	fbTcpClose: FB_SocketClose;
	bConnect: BOOL;
	bClose: BOOL;
	hTcpSock: T_HSOCKET;
	//aTcpSend:ARRAY[1..10] OF BYTE;
	//aTcpReceive:ARRAY[1..10] OF BYTE;	
	StrSend:STRING;
	StrReceive:STRING;
	fbUdpCreate:FB_SocketUdpCreate;
	hUdp: T_HSOCKET;
	bCreate: BOOL;
	port: UDINT:=60000;
	bSendTcp: BOOL;
	bReceiveTcp: BOOL;
	fbSwingHalt2: MC_Halt;
    TON01:TON;


	Lenth: UINT;
	StrSend2: STRING;
	bSendTcp2: BOOL;
	bCodeConError: BOOL;
	TON100:TON;
END_VAR




	Config();
	
	M_SendReceive();


	
	

	
	
	
	

	
	
	
	
	
	
	
	
	
	
	
	
	
	
	
	
	
(*	
   fbUdpCreate(
	sSrvNetId:= , 
	sLocalHost:= , 
	nLocalPort:= port, 
	bExecute:=bCreate , 
	tTimeout:= , 
	bBusy=> , 
	bError=> , 
	nErrId=> , 
	hSocket=> hUdp);
	
	
	*)

ACTION Config:



  IF iCode2.bComOpen THEN
	 bConnect:=TRUE;	
	 bClose:=FALSE;
	 iCode2.bComOpen:=FALSE;
  END_IF
  
   IF iCode2.bComClose THEN
	 bConnect:=FALSE;	
	 bClose:=TRUE;
	 iCode2.bComClose:=FALSE;
  END_IF 
  
  
  
fbTcpCon(
	sSrvNetId:= ''   ,          //       (*'169.254.46.193.1.1'*) , 
	sRemoteHost:='127.0.0.1'     , 
	nRemotePort:= port, 
	bExecute:=bConnect , 
	tTimeout:= , 
	bBusy=> , 
	bError=> , 
	nErrId=> , 
	hSocket=>hTcpSock );
	
fbTcpClose(
	sSrvNetId:= ''   , 
	hSocket:=hTcpSock , 
	bExecute:=bClose , 
	tTimeout:=T#5S , 
	bBusy=> , 
	bError=> , 
	nErrId=> );

IF fbTcpCon.bBusy THEN
	bConnect:=FALSE;
END_IF

IF fbTcpClose.bBusy THEN
   bClose:=FALSE;
END_IF
END_ACTION

ACTION M_SendReceive:

TON100(IN:= , PT:=T#12S , Q=> , ET=> );
  IF iCode2.bLON THEN
     StrSend:='LON16$R$N';
	 bSendTcp:=TRUE;
	 iCode2.bLON:=FALSE;
	 iCode2.bDone:=FALSE;
	 iCode2.bError:=FALSE;
	 iCode2.strCode:='';
	 Lenth:=SIZEOF(StrSend);
	 TON100.IN:=TRUE;
	// iCode.bCodeConError:=FALSE;
  END_IF

  IF iCode2.bLOFF THEN
     StrSend:='LOFF$R$N';
	 bSendTcp:=TRUE;
	 iCode2.bLOFF:=FALSE;
	 iCode2.bDone:=FALSE;
	 iCode2.bError:=FALSE;
	 iCode2.strCode:='';
	 Lenth:=SIZEOF(StrSend2);
  END_IF


fbTcpSend(
		sSrvNetId:= , 
		hSocket:=hTcpSock , 
		cbLen:=SIZEOF(StrSend), 
		pSrc:= ADR(StrSend), 
		bExecute:= bSendTcp, 
		tTimeout:= T#2S , 
		bBusy=> , 
		bError=> , 
		nErrId=> );
	
	TON01(IN:= bSendTcp, PT:= T#500MS, Q=> , ET=> );	
	IF TON01.Q THEN
		bSendTcp:=FALSE;
	END_IF
	
	
bReceiveTcp:=NOT bReceiveTcp;
fbTcpRec(
	sSrvNetId:= , 
	hSocket:= hTcpSock, 
	cbLen:=SIZEOF(StrReceive) , 
	pDest:=ADR(StrReceive) , 
	bExecute:=bReceiveTcp , 
	tTimeout:= T#5S, 
	bBusy=> , 
	bError=> , 
	nErrId=> , 
	nRecBytes=> );


(*
//IF 	StrReceive='ERROR$R0843160C8$R' OR StrReceive= 'ERROR$R' OR StrReceive='ER,' OR StrReceive=  'ERROR$R0842000C4$R' THEN
IF StrReceive<>''THEN
	IF LEN(STR:=StrReceive )>=14 AND LEN(STR:=StrReceive )<=20 AND FIND(STR1:=StrReceive , STR2:='ERROR' )=0 THEN
	  iCode2.strCode:=StrReceive;
	  StrReceive:='';
	  iCode2.bDone:=TRUE;
	ELSIF FIND(STR1:=StrReceive , STR2:='ERROR' )<>0 THEN 
	  iCode2.strCode:=StrReceive;
	  StrReceive:='';
	  iCode2.bError:=TRUE;
	END_IF
END_IF
			

IF  TON100.Q THEN
   IF StrReceive='' THEN
     // iCode.bCodeConError:=TRUE;	
   END_IF
   TON100.IN:=FALSE;
END_IF

//iCode.bCodeConError;

*)
END_ACTION

END_FUNCTION_BLOCK

// ---- POUs/BasicFunction/Motion/CS_SetpMoter.TcPOU
FUNCTION_BLOCK CS_SetpMoter
VAR_INPUT
END_VAR
VAR_OUTPUT
END_VAR
VAR
	
	
END_VAR

VAR_IN_OUT
stSetpMotor:ST_SetpMotor;//电芯出料步进电机	
END_VAR
	

VAR
iSensorCount: INT;
//R_TRIG10:R_TRIG;
//F_TRIG10:F_TRIG;
R_trig20:R_TRIG;
R_trig21:R_TRIG;
R_trig23:R_TRIG;
R_trig22:R_TRIG;
TON50:TON;
TON51:TON;
TON52:TON;
TON53:TON;
TON54:TON;
iSetp3:INT;   //电芯转移流程


END_VAR

(*********************步进电机控制*****************************)
//步进点动
stSetpMotor.bo_Up:=stSetpMotor.bJog_Up AND NOT stSetpMotor.biUpSensor ; //步进点动上升   
stSetpMotor.bo_Down:=stSetpMotor.bJog_Down AND NOT stSetpMotor.biDownSensor ;   //步进点动下降   

//步进回原点
iSensorCount:=BOOL_TO_INT(stSetpMotor.biUpSensor)+ BOOL_TO_INT(stSetpMotor.biDownSensor);
R_trig20(CLK:=stSetpMotor.bHome , Q=> );
IF R_trig20.Q  AND iSensorCount<=1 THEN
   iSetp3:=88;
   stSetpMotor.bHome:=FALSE;
   stSetpMotor.HomeDone:=FALSE;
   stSetpMotor.bPoleFull:=FALSE;
END_IF

R_trig21(CLK:=stSetpMotor.bGoWorkPos , Q=> ); //GO工作位置  
IF R_trig21.Q  THEN  //AND iSensorCount<=1
   stSetpMotor.bJog_Down:=FALSE;
   stSetpMotor.bJog_Up:=FALSE;
   iSetp3:=99;	
   stSetpMotor.HomeDone:=FALSE;
   stSetpMotor.bGoWorkPos:=FALSE;
   stSetpMotor.WorkPosDone:=FALSE;
   stSetpMotor.bPoleFull:=FALSE;
END_IF

R_trig23(CLK:=stSetpMotor.bLeaveWorkPos , Q=> ); //离开工作位置  
IF R_trig23.Q  THEN  //AND iSensorCount<=1
   stSetpMotor.bJog_Down:=FALSE;
     stSetpMotor.bJog_Up:=FALSE;
    iSetp3:=97;	
	stSetpMotor.HomeDone:=FALSE;
   stSetpMotor.bLeaveWorkPos:=FALSE;
   stSetpMotor.WorkPosDone:=FALSE;
   stSetpMotor.bPoleFull:=FALSE;
END_IF

TON50(IN:= , PT:=T#20MS , Q=> , ET=> );  //感应原点后延时
TON51(IN:= , PT:=T#20MS , Q=> , ET=> );  //对射感应原点后延时
TON52(IN:= , PT:=T#10S , Q=> , ET=> );  //感应电芯报警
TON53(IN:= , PT:=T#300MS , Q=> , ET=> );  //感
TON54(IN:=iSetp3=200 , PT:=T#20S , Q=> , ET=> );  //回原超时
R_trig22(CLK:=iSensorCount=1 , Q=> );  

IF TON54.Q THEN
	stSetpMotor.bError[1]:=TRUE;//回原超时
	stSetpMotor.bJog_Down:=FALSE;
	stSetpMotor.bJog_Up:=FALSE; 	
	iSetp3:=0;
END_IF

CASE iSetp3 OF   	
88:  
   IF stSetpMotor.biDownSensor THEN  //本来就在原点  回原完成
	   TON50.IN:=TRUE; 
	   TON52.IN:=FALSE;
	   IF TON50.Q THEN
		   stSetpMotor.HomeDone:=TRUE;
		   stSetpMotor.bJog_Down:=FALSE;
		   stSetpMotor.bJog_Up:=FALSE; 		   
		   TON50.IN:=FALSE;  
		   iSetp3:=666;   
	   END_IF
   //ELSIF  stSetpMotor.biDownSensor THEN  
	    // iSetp3:=100; 
   ELSIF  stSetpMotor.biUpSensor THEN 	   
	      iSetp3:=200;    
   ELSE                //没在任何感应 
       iSetp3:=200;    //默认往参考点回原点
   END_IF
 (* 
100:  //上升
	   stSetpMotor.bJog_Down:=FALSE;
	   stSetpMotor.bJog_Up:=TRUE;      //下限位 往上  碰到 mid2停
	    IF stSetpMotor.biRefSensor THEN
		  iSetp3:=88;	
		END_IF*)   
200:   //下降
	   stSetpMotor.bJog_Down:=TRUE;
	   stSetpMotor.bJog_Up:=FALSE; 
	   IF  R_trig22.Q THEN   //下将过程中碰到限位
		   iSetp3:=88;	 
	   END_IF   
  
(*************************对射位置***********************)   
99:    //在原位先上升    
	   stSetpMotor.bJog_Down:=FALSE;
	    stSetpMotor.bJog_Up:=TRUE;  
		TON52.IN:=TRUE;
		 iSetp3:=300;    	   
300: //对射检测
	 IF stSetpMotor.biUpSensor  THEN 
	    stSetpMotor.bJog_Down:=TRUE;
	    stSetpMotor.bJog_Up:=FALSE; 
	 END_IF

		IF stSetpMotor.biSensor   THEN //stSetpMotor.biSensor
		   TON51.IN:=TRUE; 
		   IF TON51.Q THEN 
			   stSetpMotor.WorkPosDone:=TRUE;
               stSetpMotor.bJog_Down:=FALSE;
			   stSetpMotor.bJog_Up:=FALSE; 
		       TON51.IN:=FALSE; 
			   iSetp3:=666;   
			END_IF   	
		END_IF
		
(**************************离开对射位置********************************)  		
97:     
     IF  NOT stSetpMotor.bJog_Down AND NOT stSetpMotor.bJog_Up   THEN //升降轴上升到位 
		 stSetpMotor.bJog_Down:=TRUE;
		 stSetpMotor.bJog_Up:=FALSE;
         TON53.IN:=TRUE;
		 iSetp3:=400; 
	 END_IF		
		
400:  //步进电机回原位
	     IF TON53.Q AND NOT stSetpMotor.biSensor THEN//stSetpMotor.biSensor
		   stSetpMotor.WorkPosDone:=TRUE;
		    stSetpMotor.bJog_Down:=FALSE;
		    stSetpMotor.bJog_Up:=FALSE;	 
		     TON53.IN:=FALSE;
		   iSetp3:=666; 
		 END_IF
	     IF stSetpMotor.biDownSensor  THEN
		     stSetpMotor.bJog_Down:=FALSE;
		      stSetpMotor.bJog_Up:=FALSE;	
             TON53.IN:=FALSE; 
		   // bAlarm:=TRUE;  
            stSetpMotor.bPoleFull:=TRUE;  
		    iSetp3:=666; 
		 END_IF							
END_CASE

END_FUNCTION_BLOCK

// ---- POUs/POUs/AnPart.TcPOU
PROGRAM AnPart
VAR_INPUT
          iMode                      :INT;
END_VAR

VAR
	fbAnPart: FB_UserMain;
	
END_VAR

CALL();
ACT();

ACTION ACT:
(********模切小时、天产能**********)
(*
aAnDay_date(
EE:=Q104[7],
);
*)
//运行时间统计
Antimedata(
	Month:= PLC_wMonth, 
	dDay:=PLC_wDay , 
	Hour:=PLC_wHour , 
	Mins:=PLC_wMinute , 
	Second:=PLC_wSecond , 
	Alm:=stSysState.bErrorStop AND NOT bAnDoorALM AND 
             NOT (ProductPar.AnPar.MQ.bWindSelect AND  ProductPar.parFilterAD[1].Out_Value<=ProductPar.AnPar.fDiameterAlarm_L) AND 
             NOT( NOT ProductPar.AnPar.MQ.bWindSelect AND  ProductPar.parFilterAD[2].Out_Value<=ProductPar.AnPar.fDiameterAlarm_R), 
	Wait:=(stSysState.iModehmi=2 OR  stSysState.iModehmi=3) AND (NOT stSysState.bErrorStop OR bAnDoorALM ) AND
             NOT (ProductPar.AnPar.MQ.bWindSelect AND  ProductPar.parFilterAD[1].Out_Value<=ProductPar.AnPar.fDiameterAlarm_L) AND 
             NOT( NOT ProductPar.AnPar.MQ.bWindSelect AND  ProductPar.parFilterAD[2].Out_Value<=ProductPar.AnPar.fDiameterAlarm_R) , 
	Run:=stSysState.iModehmi=1  , 
	JP_Wait:=(ProductPar.AnPar.MQ.bWindSelect AND  ProductPar.parFilterAD[1].Out_Value<=ProductPar.AnPar.fDiameterAlarm_L) OR ( NOT ProductPar.AnPar.MQ.bWindSelect AND  ProductPar.parFilterAD[2].Out_Value<=ProductPar.AnPar.fDiameterAlarm_R) , 
	Query:=MQQuery , 
	STTimedata=> , 
	date1:=MQdate );
END_ACTION

ACTION CALL:
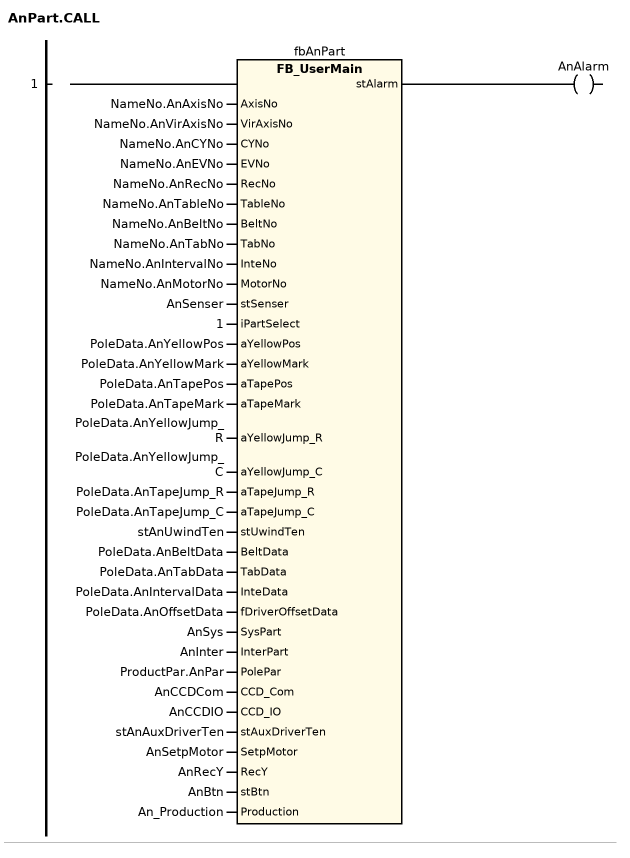
// NETWORK 1
fbAnPart(
    AxisNo := NameNo.AnAxisNo,
    VirAxisNo := NameNo.AnVirAxisNo,
    CYNo := NameNo.AnCYNo,
    EVNo := NameNo.AnEVNo,
    RecNo := NameNo.AnRecNo,
    TableNo := NameNo.AnTableNo,
    BeltNo := NameNo.AnBeltNo,
    TabNo := NameNo.AnTabNo,
    InteNo := NameNo.AnIntervalNo,
    MotorNo := NameNo.AnMotorNo,
    stSenser := AnSenser,
    iPartSelect := 1,
    aYellowPos := PoleData.AnYellowPos,
    aYellowMark := PoleData.AnYellowMark,
    aTapePos := PoleData.AnTapePos,
    aTapeMark := PoleData.AnTapeMark,
    aYellowJump_R := PoleData.AnYellowJump_R,
    aYellowJump_C := PoleData.AnYellowJump_C,
    aTapeJump_R := PoleData.AnTapeJump_R,
    aTapeJump_C := PoleData.AnTapeJump_C,
    stUwindTen := stAnUwindTen,
    BeltData := PoleData.AnBeltData,
    TabData := PoleData.AnTabData,
    InteData := PoleData.AnIntervalData,
    fDriverOffsetData := PoleData.AnOffsetData,
    SysPart := AnSys,
    InterPart := AnInter,
    PolePar := ProductPar.AnPar,
    CCD_Com := AnCCDCom,
    CCD_IO := AnCCDIO,
    stAuxDriverTen := stAnAuxDriverTen,
    SetpMotor := AnSetpMotor,
    RecY := AnRecY,
    stBtn := AnBtn,
    Production := An_Production); // FB_UserMain
AnAlarm := fbAnPart.stAlarm;
END_ACTION

END_PROGRAM

// ---- POUs/POUs/FB_UserMain.TcPOU
FUNCTION_BLOCK FB_UserMain
VAR_INPUT//输入型变量
	//Name
	AxisNo:      ST_AxisName;  //实轴名称
    VirAxisNo:      ST_VirAxisName;//虚轴名称
	CYNo:        ST_CylinderName;//气缸名称
	EVNo:        ST_ElectValveName;//阀名称
    RecNo:         ST_RecName;//纠偏名称
	TableNo:    ST_TableNo;//凸轮表名称
	BeltNo:		ST_BeltNo;//皮带工位名称
	TabNo:      ST_TabNo;//极耳工位名称
	InteNo:      ST_IntervalNo;//极耳间距工位名称	
	MotorNo:	ST_MotorName;//除尘电机名称

	stSenser:       ST_MoQieSenser;//外部光电IO
	iPartSelect:    INT;//1=正极；2=负极；

END_VAR
VAR_OUTPUT//输出型变量
	stAlarm:ST_AlarmWarn;//报警/警告汇总
END_VAR
VAR_IN_OUT//输入输出变量\
	aYellowPos:ARRAY [1..100] OF REAL;//黄标位置
	aYellowMark:ARRAY [1..100] OF BOOL;//极片黄标标志位
	aTapePos:ARRAY [1..100] OF REAL;//接带位置
	aTapeMark:ARRAY [1..100] OF BOOL;//极片接带标志位
	
	aYellowJump_R:ARRAY [1..100] OF BOOL;//极片黄标R角跳切标志
	aYellowJump_C:ARRAY [1..100] OF BOOL;//极片黄标裁切跳切标志
	aTapeJump_R:ARRAY [1..100] OF BOOL;//极片接带R角跳切标志
	aTapeJump_C:ARRAY [1..100] OF BOOL;//极片接带裁切跳切标志
	
	stUwindTen:ST_Tension;//放卷张力
	BeltData:ARRAY[1..40]   OF  ST_BeltData;//皮带数据 (裁断后)
	TabData:ARRAY[1..20]   OF  ST_TabData;//极耳数据 (裁断前)
	InteData:ARRAY[1..20]   OF  ST_IntervalData;//极耳间距数据 (裁断前)
	fDriverOffsetData     :ARRAY [1..50] OF REAL;//主驱补偿量记录
	SysPart:ST_SystemPart;//正负区分(系统)
	InterPart:ST_P2InteractPart;//正负区分(交互)
	PolePar:ST_ParProduct;//工艺参数
	CCD_Com:ST_CCDCom;//通讯时使用
	CCD_IO:ST_CCDIO;//CCD拍照信号
//	stUwindLTen:ST_Tension;//张力左放卷
//	stUwindRTen:ST_Tension;//张力右放卷
	stAuxDriverTen:ST_Tension;//张力辅驱	
	SetpMotor:ST_SetpMotor;//NG排杆电机
	RecY:ST_RecY;//模具Y纠偏
	stBtn:			ST_MoQieButton;//外部按钮和按钮灯
	Production:LocalProduction;//产能
END_VAR
VAR//内部变量
//
	RecYRules:ARRAY [1..5] OF BOOL;//不纠偏条件
//新增
	rYellowPosRel:REAL;//黄标感应器相对于极耳位置的差
	rYellowJumpPos1:REAL;//黄标跳切区间判断位置1
	rYellowJumpPos2:REAL;//黄标跳切区间判断位置2


	//Init
		rtInit   : Tc2_Standard.R_TRIG;
		iInitStep:INT;
		tonInit: ARRAY [1..10] OF TON;
	//CamCall
		fbVirBeltCam:FB_CamMQBeltV1;
		fbNGPushCam:FB_CamMQPushV1;
		fbMouldCam:FB_CamMQPushV2;		
		fbCuterCam:FB_CamMQPushV2;
		fbDriverCam:FB_CamMQDriverV1;
		fbVDriverCam:FB_CamVirDriver;
		
		fbCCDPressCam:FB_CamMQCCDPressV1;
		fbPoleBufferCam:FB_CamPoleBuffer;
		fbPoleBufferCam_1:FB_CamPoleBuffer_1;

		stPoleBufferCam:ST_Cam;
		stPoleBufferCam_1:ST_Cam;
		stVirBeltCam:ST_Cam;
		stNGPushCam:ST_Cam;
		stCuterCam:ST_Cam;
		stDriverCam:ST_Cam;
		stVirDriverCam:ST_Cam;
		stBufferTen: ST_TenBuffer;
		stMouldCam:ST_Cam;
		stCCDPressCam:ST_Cam;
	//MoTionManual
		fbRotateSwitchCode:FB_RotateSwitchCode;
		rtMotionBtn   :ARRAY[1..20] OF  Tc2_Standard.R_TRIG;
		ftMotionBtn   :ARRAY[1..20] OF  Tc2_Standard.F_TRIG;
		rtPoleBtn:Tc2_Standard.R_TRIG;
		ftPoleBtn:Tc2_Standard.F_TRIG;
	//CyManual
		rtCyBtn   :ARRAY[1..20] OF  Tc2_Standard.R_TRIG;
		ftCyBtn   :ARRAY[1..20] OF  Tc2_Standard.F_TRIG;
	//GearCall
		//fbVirDriverGear:FB_GearInDyn;
		fbCuterBeltGear:FB_GearInDyn;
		fbNGReverseBeltGear:FB_GearInDyn;
		fbDedustBeltGear:FB_GearInDyn;
		fbDedustReverseBeltGear:FB_GearInDyn;
		fbSubBelt1Gear:FB_GearInDyn;
		fbSubBelt2Gear:FB_GearInDyn;
		fbSubBelt3Gear:FB_GearInDyn;
		
		//stVirDriverGear:ST_Gear;
		stCuterBeltGear:ST_Gear;
		stNGReverseBeltGear:ST_Gear;
		stDedustBeltGear:ST_Gear;
		stDedustReverseBeltGear:ST_Gear;	
		stSubBelt1Gear:ST_Gear;
		stSubBelt2Gear:ST_Gear;
		stSubBelt3Gear:ST_Gear;

	//TensionCall
		fbUwindTen:FB_TensionPole_1;//放卷张力
	
		//fbUwindLTen:FB_TensionPole;
		//fbUwindRTen:FB_TensionPole;
		fbAuxDriverTen:FB_TensionV3;
		fbTorqueControl:MC_TorqueControl;
	//Home
		iHomeStep:INT;
		tonHome: ARRAY [1..10] OF TON;
		rtHome   :ARRAY[1..5] OF  Tc2_Standard.R_TRIG;
	//FunctionTen
		iTensionStep:INT;
		tonTension: ARRAY [1..10] OF TON;
		rtTension   :ARRAY[1..5] OF  Tc2_Standard.R_TRIG;
		bMethodTenBufferEnable:BOOL;//自动上张力
		bMethodTenBufferDisEnable:BOOL;//自动解除张力
	//FunctionCam
		iCamStep:INT;
		tonCam: ARRAY [1..10] OF TON;
		rtCam   :ARRAY[1..5] OF  Tc2_Standard.R_TRIG;
		bMethodCamEnable:BOOL;//自动上凸轮
		bMethodCamDisEnable:BOOL;//自动解除凸轮
	//Condition
		rtbtnRest   :  Tc2_Standard.R_TRIG;
		rtCondition: ARRAY [1..10] OF Tc2_Standard.R_TRIG;
		rtCount1: Tc2_Standard.R_TRIG;
		rtCount2: Tc2_Standard.R_TRIG;
		tonCondition: ARRAY [1..50] OF TON;
		bAutoReadyTemp1:BOOL;//张力准备好
		bAutoReadyTemp2:BOOL;//凸轮创建OK
		bAutoReadyTemp3:BOOL;//设备状态
		bAutoReadyTemp4:BOOL;//轴准备好
		bAutoReadyTemp5:BOOL;//轴没有报警
		iPoleNoHave:INT:=2;//无料统计(主轴可连续运行标志)
		iPoleNoHaveA:INT:=2;//无料统计1(主轴可连续运行标志)
		iPoleCarryEver:INT:=3;//手动时切换 1=极片仅流至1号；2=极片可流至2号;3=极片流至末端
		iMainMode:INT:=0;//皮带耦合状况  1=停止等待；2=自由模式；
		bBelt_1:ARRAY [1..3] OF BOOL;//皮带末倒数第1位有料  1=1号分段皮带 2=2号分段皮带 3=3号分段皮带
		bBelt_2:ARRAY [1..3] OF BOOL;//皮带末倒数第2位有料  1=1号分段皮带 2=2号分段皮带 3=3号分段皮带
		//bP2M3Need:BOOL;//3号叠台要料
		//bP2AllNoNeed:BOOL;//三个叠台都不要料
		i2:INT;
		bTest: ARRAY [1..20] OF BOOL;//测试用
		MA10: BOOL;
		fTagatTime: REAL;		
	//AUTO
	    fbTailCurl:FB_TailCurl_PID;
		fbRectifyGM:FB_RectifyGM;
		iAutoRunStep:INT;//主流程
		iAutoAuxStep1:INT;//辅助流程:凸轮
		iAutoAuxStep2:INT;//辅助流程:张力
		iAutoAuxStep3:INT;//辅助流程:尺寸检测
		iAutoAuxStep4:INT;//辅助流程:冲R角定位检测
		iAutoAuxStep5:INT;//辅助流程:裁切定位检测
		iAutoAuxStep6:INT;//辅助流程:1#取料
		iAutoAuxStep7:INT;//辅助流程:2#取料
		iAutoAuxStep8:INT;//辅助流程:3#取料
		iAutoAuxStep9:INT;//辅助流程:取片信号交互
		iAutoAuxStep10:INT;//辅助流程:CCD标定
		iAutoAuxStep11:INT;//辅助流程:线扫结果
		//iAutoAuxStep11:INT;//辅助流程:蓝胶检测
		//iAutoAuxStep12:INT;//辅助流程:
		//iAutoAuxStep13:INT;//辅助流程:
		//iAutoAuxStep14:INT;//辅助流程:
		//iAutoAuxStep15:INT;//辅助流程:
		tonAuto: ARRAY [1..40] OF TON;
		rtAuto   :ARRAY[1..20] OF  R_TRIG;
		ftAuto   :ARRAY[1..20] OF  f_TRIG;
		bFlgStoping:BOOL;//主轴ABS停止中
		bSysStoping:BOOL;//系统停止中
		//bMA10:BOOL;
		//bMA11:BOOL;
		//bMA12:BOOL;
		//bMA20:BOOL;
		bMA21:BOOL;
		//bMA22:BOOL;
		//bMA30:BOOL;
		bMA31:BOOL;
		//bMA32:BOOL;
		//bMA40:BOOL;
		//bMA41:BOOL;
		//bMA42:BOOL;
		//bMA50:BOOL;
		//bMA51:BOOL;
		//bMA52:BOOL;
		bFristPole:BOOL;//首张极片标志
		bPeaceBelt1Front:BOOL;//1#取料工位前有料
		bPeaceBelt2Front:BOOL;//2#取料工位前有料
		bPeaceBelt3Front:BOOL;//3#取料工位前有料
		bHavePeaceBelt:BOOL;//皮带上有料
		iBeltNoPeaceCount:INT;//皮带上无片工位计数
		bBelt2Need:BOOL;//皮带2要料
		bBelt3Need:BOOL;//皮带3要料
		//fSubBeltMasterScaling:LREAL;//
		//fNGPushMasterScaling:LREAL;//备用
		//fTakeCyDegree:LREAL;//取料时最短气控动作角度
		//fTakeAxisDegree:LREAL;//取料时最短电机动作角度
		fRecordOverHangInMainPos:LREAL;//记录主轴位置
		fRecordOverHangInMainPosMod:LREAL;//记录主轴模数位置
		fRecordMouldCCDInMainPos:LREAL;//记录主轴位置
		fRecordMouldCCDInMainPosMod:LREAL;//记录主轴模数位置
		fRecordCuterCCDInMainPos:LREAL;//记录主轴位置
		fRecordCuterCCDInMainPosMod:LREAL;//记录主轴模数位置
		//bTakePolePushMode:BOOL;//TRUE 升降取片
		//bTakePoleAirSign:BOOL;//吹气取片标志
		//bTakeSubBelt1Sign:BOOL;//等待1号皮带耦合中
		//bTakeSubBelt2Sign:BOOL;//等待2号皮带耦合中
		//bTakeSubBelt3Sign:BOOL;//等待3号皮带耦合中
		//bCamInAbsSign:BOOL;//倒吸耦合主轴ABS
		i:INT;
		i1:INT;
		i3:INT;
		i4:INT;
		i5:INT;
		i6:INT;
		i7:INT;
		i8:INT;
		i9:INT;	
		i10:INT;
		i11:INT;
		i12:INT;
		i13:INT;
		i14:INT;
		i15:INT;
		i16:INT;
		i17:INT;
		i18:INT;
		i19:INT;
		i20:INT;
		i21:INT;
		bBelt1Gearask:BOOL;//皮带1耦合请求
		bBelt2Gearask:BOOL;//皮带2耦合请求
		bBelt3Gearask:BOOL;//皮带3耦合请求
		bBelt1Taking:BOOL;//1号皮带取料流程中
		bBelt2Taking:BOOL;//2号皮带取料流程中
		bBelt3Taking:BOOL;//3号皮带取料流程中
		fOffsetDeg	: ARRAY [1..10] OF REAL;
		fTabInteM_1:REAL;//模具前一个工位极耳间距
		fTabInteM_2:REAL;//测试用，模具前一个工位极耳间距///
		fDriverOffset1:REAL;//主驱补偿量辅助1
		fDriverOffset2:REAL;//主驱补偿量辅助2
		fDriverOffset3:REAL;//主驱补偿量辅助3
		fDriverOffset4:REAL;//主驱补偿量辅助4
		fDriverOffset5: REAL;	//主驱补偿量辅助5
		fDriverOffset6: REAL;	//主驱补偿量辅助6
		fDriverOffset7: REAL;	//主驱补偿量辅助7   以肩宽为基准
		//fMouldXOffset1:REAL;//模具X补偿量辅助1
		//fMouldXOffset2:REAL;//模具X补偿量辅助2
		//fMouldXOffset3:REAL;//模具X补偿量辅助3
		//fMouldXOffset4:REAL;//模具X补偿量辅助4
		fMouldXOffset7:REAL;//模具X补偿量辅助7  以肩宽为基准
    	fMouldXOffset8:REAL;//模具Y补偿量辅助7  \
		fBluePos:ARRAY [1..20] OF REAL;//蓝胶位置
		fLineScanPos:ARRAY [1..20] OF REAL;//线扫NG位置
		iNGPoleCount:INT;//NG极片计数
		iNGPoleCount1:INT;//NG极片计数
		fDegreeRec1:REAL;//角度纠偏  方差值
		fDegreeRec2:REAL;//角度纠偏  均值
		bJumpCut:BOOL;//跳切标记
		iNormalCuter:INT;//正常裁断计数
		iMouldRunTableSel:UINT;//模具当前周期的凸轮选择
		iCuterRunTableSel:UINT;//裁切当前周期的凸轮选择
		bChaNoPhoto: BOOL;//标定时，冲R角CCD相机不拍照
		bCutNoPhoto: BOOL;//标定时，裁切CCD相机不拍照
		bSubBelt1fratio:BOOL;//FALSE=分段皮带1比例为0
		bSubBelt2fratio:BOOL;//FALSE=分段皮带2比例为0
		bSubBelt3fratio:BOOL;//FALSE=分段皮带3比例为0
		itest: INT; // 1: 静止绝对   2：运动绝对  3:触发速度   4：立即停止   0：无效值
		iPoleNoHave1: INT;//运动耦合时记录料况
		iPoleNoHave2: INT;//静止耦合时记录料况
		  fbAuxDriverTen2     : FB_GearInMulti;
		  fbTensionVirDriver     : FB_TensionVirDriver;
		 fM_TabInterData    :ARRAY [1..50] OF REAL;//倒角计算极耳间距记录
		 fPoleWithOffset:REAL;//实时补偿量
		 iNGSize:INT:=0;//尺寸NG计数 	
         iNGScane:INT:=0;//线扫检测连NG计数 	
		bEnable: BOOL;
		bEnable2: BOOL;
		ftest1: REAL;
		ftest2: LREAL;
		ftest3: LREAL;
		iAutoRunStep20: INT;
		itest1: INT;
		itest2: INT;
		itest3: INT;
		itest4: INT;	
		fMouldX_Offset: REAL;
		bPoleBufferSel:BOOL;//FALSE=凸轮切换为正常凸轮；True=凸轮切换为高速凸轮
		fPoleBufferCompensation:REAL:=0;
		bFindTab:BOOL;//找极耳标志
	//ClearBeltAUTO
		iClearBeltStep:INT;
		tonClearBelt: ARRAY [1..10] OF TON;
		rtClearBelt   :ARRAY[1..5] OF  Tc2_Standard.R_TRIG;	
		rtMouldClear1   :Tc2_Standard.R_TRIG;    //模具切刀计数清零
		rtMouldClear2   :Tc2_Standard.R_TRIG;    //模具切刀计数清零
		rtCuterClear   :Tc2_Standard.R_TRIG;     //模具裁切切刀计数清零
		MQ_alarm_ton :ARRAY[1..40] OF TON;
	bBelt_NO1: BOOL;
	bBelt_NO2: BOOL;
	bBelt_NO3: BOOL;
	ab: INT;
	
		bBelt1Need: BOOL;
	bBeltStatusUpData: BOOL;
	iBeltNeedAlarm: INT;
	iBeltNeedAlarm3: INT;
	iBeltNeedAlarm10: INT;
	iBeltNeedAlarm5: INT;
	iCount1: DINT;
	iCount2: DINT;
	iCount3: DINT;
	DelayM1: TON;
	iPeaceAlarmCount1: DINT;
	iPeaceAlarmCount2: DINT;
	iPeaceAlarmCount3: DINT;
	iPeaceMoveAlarm1: INT;
	iPeaceMoveAlarm2: DINT;
	rtVirMainCount: R_TRIG;
	iVirMainCycleCount: DINT;
	iVirMainCycleCountTemp1: DINT;
	iVirMainCycleCountRel: DINT;
	iPeaceAlarmCount1Temp: DINT;
	iPeaceAlarmCount1Rel: DINT;
	iPeaceAlarmCount2Temp: DINT;
	iPeaceAlarmCount2Rel: DINT;
	iPeaceAlarmCount3Temp: DINT;
	iPeaceAlarmCount3Rel: DINT;
	bBelte1PeaceAlarm: BOOL;
	bBelte2PeaceAlarm: BOOL;
	bBelte3PeaceAlarm: BOOL;
	DelayStep6: TON;
	rtPeaceMoveAlarm: R_TRIG;
	bMA15: BOOL := TRUE;
	iStopCount: INT;
	iAutoAuxStep6Temp: INT;
	iOverCycleCount1: INT;
	iAutoAuxStep7Temp: INT;
	iAutoAuxStep8Temp: INT;
	iOverCycleCount2: INT;
	iOverCycleCount3: INT;
	
	rtMQDriverOnce: R_TRIG;	
	
	
	
	iMQDriverOnceSetp1: INT;
	rtEarCheck1: R_TRIG;
	rtMQCutOnce: R_TRIG;
	iP1MQCutOnce: INT;
	ttLinePhoto: R_TRIG;
	fRecordLineineScanCCDInMainPos: LREAL;
	fRecordLineineScanCCDInMainPosMod: REAL;
	XianSaong: ARRAY [0..20] OF INT;
	XianSaong1: ARRAY [0..20] OF INT;
	XianSaong_Up: ARRAY [0..20] OF INT;
	XianSaong_Down: ARRAY [0..20] OF INT;		
	CutMark_R: ARRAY [0..10] OF BOOL;///没有检测到极耳时跳切
	iCount10: DINT;
	//t_Time:Tc2_Standard.TON;
		CCD_Rounde: FB_CCD_Rounde;
	rtBelt1TakingReset1: R_TRIG;
	rtBelt1TakingReset2: R_TRIG;
	rtBelt1TakingReset3: R_TRIG;
	rtNGPush: R_TRIG;
	iNGStep: INT;
	
   fbPoleBufferTen   :   FB_TensionBuffer;
	NG_Sum: INT;
	YellowmarkNG :ARRAY[1..10] OF INT ;//裁切前黄标NG
	aAq1: BOOL;
	aAq2: BOOL;
	
	
//新增备用
	rMQUse:ARRAY[1..20] OF R_TRIG;//模切上升沿
	fMQUse:ARRAY[1..20] OF F_TRIG;//模切下降沿
	tMQUse:ARRAY[1..20] OF TON;//模切定时器	
	fAveWidth: REAL;// 平均计算片宽
	iMainVel:UINT:=10;  //设置速度 PPM (最小值1,最大值200) 
	nInt:ARRAY [1..10] OF UINT:=[30];//
	bDTSyn:BOOL;//叠台同步
	bFirstCylce:BOOL;
	NGBox: INT;
	
	aYellowPos_R:ARRAY [1..100] OF REAL;//黄标位置
	aYellowPos_R2:ARRAY [1..25] OF REAL;//黄标到裁切刀的距离
	aTapePos_R2:ARRAY [1..25] OF REAL;//的距离
	aYellowPos_RC: REAL;//黄标位置
	aYellowPos_C:ARRAY [1..100] OF REAL;//黄标位置
	Test:BOOL;//
	DemarcateStep:UINT;//初始卷径标定自动步

	
	
	
	bRectifyTest: BOOL;
	fCyDDRActPos:LREAL;//设备自动时记录主驱当前位置mm
	bCyDDRMark:BOOL;//设备自动时纠偏启动标志位
	rtBoardPressTurn: R_TRIG;
	rtBreakError: R_TRIG;
	rtRecManual1: R_TRIG;
	rtRecManual2: R_TRIG;
	
	RecSetp: INT;
	bFlgRecManual: BOOL;
	bFlgRecAuto: BOOL;
	bFlgRecCenter: BOOL;
	iRecStatus: INT;
	tonRecCenterDelay: TON;
	bRecCenterMoving: BOOL;
	tonRecDelay: TON;
	
		iTabOffsetStep: INT;
	rtTabSenser: R_TRIG;
	ftTabSenser: F_TRIG;
	bRecordPosM1: BOOL;
	bRecordPosM2: BOOL;
	fVirMainSenserPos1: REAL;  //极耳上升沿记录主虚轴位置
	fVirMainSenserPos2: REAL; //极耳下降沿记录主虚轴位置
	fReadDriverPos1: REAL;//读取极耳上升沿主驱凸轮表位置
	arrfReadDriverPos1: ARRAY[1..50] OF REAL; //记录极耳上升沿主驱凸轮表位置
	arrfReadDriverPos2: ARRAY[1..50] OF REAL;//记录极耳下降沿主驱凸轮表位置
	K1: INT := 1;
	fReadDriverPos2: REAL;//读取极耳下降沿主驱凸轮表位置
	fTabWidth: REAL;//极耳标准宽
	fCalueTabWidth: REAL;//计算极耳宽度
	fDriverStanderBasePos: REAL;//极耳下降沿基准主驱凸轮位置
	fTabOffset: REAL; 
	bDriverStanderBasePosEN: BOOL;  //极耳大范围调整屏蔽
	bFlgTabPosOver: BOOL;//极耳位置超限标志  给Auto4用
	fDriverOffset: REAL;  //极耳位置偏移量  给Auto4用
	fbReadTabCamSlavePos :Tc2_MC2_Camming.MC_ReadCamTableSlaveDynamics;////
	
	
	iCount100: DINT;
	iCount101: DINT;
	
	iTabWidth_JS: INT;

	iStopCount2: DINT;
	iStopCount3: INT;
	iStopCount4: INT;
	UnWind_L: INT;
	
	bLineScanResult1_UP: BOOL;
	bLineScanResult2_UP: BOOL;
	bLineScanResult1_Down: BOOL;
	bLineScanResult2_Down: BOOL;
	rLineScanOK_UP: R_TRIG;
	rLineScanNG_UP: R_TRIG;
	rLineScanOK_Down: R_TRIG;
	rLineScanNG_Down: R_TRIG;
	r1aser:ARRAY[0..7] OF R_TRIG;
	
	 fDA1: REAL;
	fDA2: REAL;
	bFlgLineScanOver: BOOL;
	rLineScan_UPTCP: R_TRIG;
	rLineScan_DownTCP: R_TRIG;
	
				//4连黄标尾料检测  SJ
		rtTabSenser2: R_TRIG;
		ftTabSenser2: F_TRIG;
    	iEndYellowMackStep: INT;	
		arrbRecordPos:  ARRAY[1..4] OF   BOOL;  //记录黄标下降沿标志
	 	fbReadTabCamSlavePos2 :Tc2_MC2_Camming.MC_ReadCamTableSlaveDynamics;////
		arrfVirMainSenserPos:       ARRAY[1..4] OF  LREAL;  //黄标下降沿主虚轴位置
	    K2: INT;
	    fD12:    REAL;   //黄标1与黄标2 的间距
	    fD23:    REAL;  //  //黄标2与黄标3的间距
	    fD34:    REAL;    //黄标3与黄标4的间距
		
	
	  bYellowMackAlarm: BOOL;
	
	
	
	aYellowPosTemp1: LREAL;
	bYellowPosTemp1: BOOL;
	aYellowPosTemp2: LREAL;
	bYellowPosTemp2: BOOL;

	bAnLaser:BOOL;
	bCaLaser:BOOL;

	fSumDriverOffsetData: REAL;
	fArvDriverOffsetData: REAL;
	bMA1: BOOL;
	fTab_OffsetC: REAL;
	
	
	iFlgCompCount: INT;
	iCompCount: INT;
	iRTransCompCount: INT:=1;//R角横深补偿次数
	arrOffset :ARRAY[0..20] OF REAL;	
	i30: INT;
	iCount20: DINT;
	fSumTransverData: REAL;//R角横深求和
	fArvTransverData: REAL;//R角横深平均值
	iNGState:INT;//踢废状态
	bFourYellowFlg:BOOL;	
	bYellowPosTemp3: BOOL;
	bYellowPosTemp4: BOOL;
	bYellowPosTemp5: BOOL;
	bYellowPosTemp6: BOOL;
	fBelt1Pos:ARRAY [0..10] OF LREAL;
	fBelt2Pos:ARRAY [0..10] OF LREAL;
	fBelt3Pos:ARRAY [0..10] OF LREAL;
	
	fSumTransverData2: REAL;//R角纵深求和
	fArvTransverData2: REAL;//R角纵深平均值
	iRTransCompCount2: INT:=1;//R角横深补偿次数
	fRSizeBase  :REAL;
	 K3: INT;
	bComMode: BOOL;
	
	K4: INT;
	
	tonBtn: ARRAY [1..10] OF TON;
	
	arrModPos: ARRAY[1..500] OF STRING(50);
	K10: INT:=1;		

	bMA10: BOOL;
	bTapeMark: BOOL;//接带标志
	aTapepos2: LREAL;//接带后
	bSubBelt1Alarm1: BOOL;
	bSubBelt1Alarm2: BOOL;
	bSubBelt2Moving1 : BOOL;
	bSubBelt2Moving2 : BOOL;
	bSubBelt3Moving1 : BOOL;
	bSubBelt3Moving2 : BOOL;
    iRuningFlg: INT;
	
END_VAR
VAR PERSISTENT
		fDriverDDRActPos:REAL;//主驱动当前位置(mm)	
		
		fLugActPos: REAL;//极耳位置记录
		bLugActPosMark_r:BOOL;//上升沿极耳位置已记录标志位
		bLugActPosMark_f:BOOL;//下降沿极耳位置已记录标志位
		bYellowActPosMark:BOOL;//黄标位置已记录标志位
		fYellowMarkActPos: REAL;//黄标位置记录
		bYellowMark:ARRAY[1..50] OF BOOL;//极片黄标标志-----切刀到黄标感应器直接极片个数
		aFB_ProductionDataLocal:FB_ProductionDataLocal;
		pRollWind:POINTER TO AXIS_REF;//放卷轴指针
		
END_VAR

CASE stSysState.iMode OF
0:
     F09INIT();
   
1://自动
   F0500MainAuto();
   F0501MainAuto1();
   F0502MainAuto2();
   F0503MainAuto3();
   F0504MainAuto4();
   F0505MainAuto5();
   F0506MainAuto6();
3://手动
   F00Home();
   F01MotionManual();
   F02CylinderManual();
   F09INIT();
   F13ClearBelt();
4://停止
;
END_CASE
F10GearCall();
F11CamCall();
F12TensionCall();
F03FunctionTen();
F04FunctionCam();
F05Rectifydev();
F07Condition();
F0511CCDAuto();
F0512CarryAuto();
F0599AutoAux();
Alarm();
Product();

ACTION Alarm:

/////////凸轮创建报警/////////
stAlarm.arrCreatTableAlarm[1]:=stPoleBufferCam.bCreatTableError OR stPoleBufferCam_1.bCreatTableError;//极片缓存电机创建凸轮报警
stAlarm.arrCreatTableAlarm[2]:=stDriverCam.bCreatTableError;//主驱动电机创建凸轮报警
stAlarm.arrCreatTableAlarm[3]:=stMouldCam.bCreatTableError;//模具切刀电机创建凸轮报警
stAlarm.arrCreatTableAlarm[4]:=stCuterCam.bCreatTableError;//裁切切刀电机创建凸轮报警
stAlarm.arrCreatTableAlarm[5]:=stCCDPressCam.bCreatTableError;//CCD压片升降电机创建凸轮报警
stAlarm.arrCreatTableAlarm[6]:=stVirBeltCam.bCreatTableError;//皮带虚轴电机创建凸轮报警
//stAlarm.arrCreatTableAlarm[7]:=stNGPushCam.bCreatTableError;//NG踢料电机创建凸轮报警

/////////凸轮耦合报警/////////
stAlarm.arrCamInAlarm[1]:=stPoleBufferCam.bError OR stPoleBufferCam_1.bError;//极片缓存电机凸轮耦合报警
stAlarm.arrCamInAlarm[2]:=stDriverCam.bError;//主驱动电机凸轮耦合报警
stAlarm.arrCamInAlarm[3]:=stMouldCam.bError;//模具切刀电机凸轮耦合报警
stAlarm.arrCamInAlarm[4]:=stCuterCam.bError;//裁切切刀电机凸轮耦合报警
stAlarm.arrCamInAlarm[5]:=stCCDPressCam.bError;//CCD压片升降电机凸轮耦合报警
stAlarm.arrCamInAlarm[6]:=stVirBeltCam.bError;//皮带虚轴电机凸轮耦合报警
//stAlarm.arrCamInAlarm[7]:=stNGPushCam.bError;//NG踢料电机凸轮耦合报警

/////////张力报警/////////
stAlarm.arrTenAlarm[1]:=stUwindTen.bError AND PolePar.MQ.bWindSelect;//左放卷张力报警
stAlarm.arrTenAlarm[2]:=stUwindTen.bError AND NOT PolePar.MQ.bWindSelect;//右放卷张力报警
stAlarm.arrTenAlarm[3]:=stAuxDriverTen.bError;//辅驱张力报警
stAlarm.arrTenAlarm[4];//前摆杆张力电机张力报警
/////////齿轮报警/////////
//stAlarm.arrGearAlarm[1]:=stVirDriverGear.bError;//虚拟放卷电机齿轮报警
stAlarm.arrGearAlarm[2]:=stCuterBeltGear.bError;//裁切输送皮带电机齿轮报警
stAlarm.arrGearAlarm[3]:=stNGReverseBeltGear.bError;//踢废倒装皮带电机齿轮报警
stAlarm.arrGearAlarm[4]:=stDedustBeltGear.bError;//上表面除尘皮带电机齿轮报警
stAlarm.arrGearAlarm[5]:=stDedustReverseBeltGear.bError;//下表面除尘倒装皮带电机齿轮报警
stAlarm.arrGearAlarm[6]:=stSubBelt1Gear.bError;//分段主皮带1电机齿轮报警
stAlarm.arrGearAlarm[7]:=stSubBelt2Gear.bError;//分段主皮带2电机齿轮报警
stAlarm.arrGearAlarm[8]:=stSubBelt3Gear.bError;//分段主皮带3电机齿轮报警
/////////流程报警/////////
stAlarm.arrFlowAlarm[1];//自动已占用    料盒排杆电机去工作位超时
stAlarm.arrFlowAlarm[2];	//极片放卷按钮盒急停已按下
stAlarm.arrFlowAlarm[3];	//NG料盒按钮盒急停已按下
stAlarm.arrFlowAlarm[4];	//面板急停已按下
stAlarm.arrFlowAlarm[5];	//外罩急停1处已按下
stAlarm.arrFlowAlarm[6];	//外罩急停2处已按下
stAlarm.arrFlowAlarm[7];	//外罩急停3处已按下
stAlarm.arrFlowAlarm[8];	//线扫CCD软件心跳超时
stAlarm.arrFlowAlarm[9];	//外罩门禁1已开
stAlarm.arrFlowAlarm[10];	//外罩门禁2已开
stAlarm.arrFlowAlarm[11];	//外罩门禁3已开
stAlarm.arrFlowAlarm[12];	//外罩门禁4已开
stAlarm.arrFlowAlarm[13];	//外罩门禁5已开
stAlarm.arrFlowAlarm[14];	//面阵CCD软件心跳超时
stAlarm.arrFlowAlarm[15];	//左极片料卷已用完，请停机处理！
stAlarm.arrFlowAlarm[16];	//右极片料卷已用完，请停机处理！
//stAlarm.arrFlowAlarm[17]:=SetpMotor.bError[1];	//料盒排杆电机回原超时，请查看！
stAlarm.arrFlowAlarm[18];	//放卷纠偏故障
stAlarm.arrFlowAlarm[19];	//过程纠偏故障
stAlarm.arrFlowAlarm[20];   //连续尺寸NG，请报警处理
stAlarm.arrFlowAlarm[21];   //CCD尺寸检测出无片，请查看是否堵片。
stAlarm.arrFlowAlarm[22]:=RecY.bError AND NOT ProductPar.iModeEN.bEmptyRunEN AND NOT ProductPar.iModeEN.bMouldYRecEN;//   模具Y纠偏    报错
stAlarm.arrFlowAlarm[23];//分段皮带堵片报警
//stAlarm.arrFlowAlarm[24];//线扫NG报警
stAlarm.arrFlowAlarm[25];//上线扫超时报警
stAlarm.arrFlowAlarm[26];//在设定的时间内，正极模切NG数大于NG报警个数，检查模切异常后，复位启动。
stAlarm.arrFlowAlarm[27];//下线扫超时报警
stAlarm.arrFlowAlarm[28];	//Event 547
stAlarm.arrFlowAlarm[29];	//Event 548
stAlarm.arrFlowAlarm[30];	//模切主驱动位置错误，请手动复位。
stAlarm.arrFlowAlarm[31];	//分段皮带1取料位置异常。
stAlarm.arrFlowAlarm[32];	//分段皮带2取料位置异常。
stAlarm.arrFlowAlarm[33];	//分段皮带3取料位置异常。
stAlarm.arrFlowAlarm[34];	//Event 553
stAlarm.arrFlowAlarm[35];	//裁切切刀堵料，请人工清理后开机！！！-------------暂时屏蔽
stAlarm.arrFlowAlarm[36];	//堵料感应器异常，请检查感应器是否损坏；
stAlarm.arrFlowAlarm[37];	//NG片踢废失败报警，请检查并把NG片拿掉-------------暂时屏蔽
stAlarm.arrFlowAlarm[38];	//踢废失败感应器未检测到极片，请确认感应器是否安装正确；-------------暂时屏蔽
stAlarm.arrFlowAlarm[39];//NG料盒料满报警
stAlarm.arrFlowAlarm[40];	//极片极耳超出CCD检测范围
stAlarm.arrFlowAlarm[41];	//极片来料不良，请检查
stAlarm.arrFlowAlarm[42];	//当前料卷检测到四连标
stAlarm.arrFlowAlarm[43];	//分段皮带3料盒满料报警
stAlarm.arrFlowAlarm[44];	///NG踢废堵料报警
stAlarm.arrFlowAlarm[45];	//线扫检测连续NG多少片后，报警
stAlarm.arrFlowAlarm[46];	//Event 565
stAlarm.arrFlowAlarm[47];	//Event 566
stAlarm.arrFlowAlarm[48];	//Event 567
stAlarm.arrFlowAlarm[49];	//Event 568
stAlarm.arrFlowAlarm[50];	//Event 569

/////////提示////////
stAlarm.arrLightWarn[1];//自动已占用   冲R角CCD定位检测NG，请查看！
stAlarm.arrLightWarn[2];//自动已占用	冲R角CCD定位检测超时，请查看！		
stAlarm.arrLightWarn[3];//自动已占用    裁切CCD定位检测NG，请查看！
stAlarm.arrLightWarn[4];//自动已占用    裁切CCD定位检测超时，请查看！		
stAlarm.arrLightWarn[5];//自动已占用    尺寸CCD检测超时，请查看！
stAlarm.arrLightWarn[6];//自动已占用     模具前CCD检测计算极耳间距异常！
stAlarm.arrLightWarn[7];//自动已占用     主驱补偿量超过半个片宽，请查看！
stAlarm.arrLightWarn[8];//自动已占用     模具X补偿量超过纠偏电机行程
stAlarm.arrLightWarn[9];//自动已占用     裁切角度纠偏量超过纠偏电机行程
stAlarm.arrLightWarn[10] ;//   空
stAlarm.arrLightWarn[11] ;// 自动已占用    皮带运行出现记忆紊乱，请查看！
stBtn.NGBoxStartLight:=stAlarm.arrLightWarn[12] AND fbPulseCtrl[4].Q;// NG料盒已满
stAlarm.arrLightWarn[13];// NG料盒未到位
stAlarm.arrLightWarn[14];//左极片料卷即将用完！
stAlarm.arrLightWarn[15];//右极片料卷即将用完！
stAlarm.arrLightWarn[16];//备用
stAlarm.arrLightWarn[17];//备用
stAlarm.arrLightWarn[18];//主轴定位运算警告
stAlarm.arrLightWarn[19];//模具纠偏X轴定位运算警告
stAlarm.arrLightWarn[20];//裁切角度纠偏轴定位运算警告
stAlarm.arrLightWarn[21];//NG1轴定位运算警告
stAlarm.arrLightWarn[22];//线扫NG警告
stAlarm.arrLightWarn[23];//倒装皮带被抬起，请拿走倒装皮带的首尾两块极片
stAlarm.arrLightWarn[24];//分段皮带1有极片无极片编号提示
stAlarm.arrLightWarn[25];//分段皮带2有极片无极片编号提示
//NG料盒满料报警
IF tonAuto[23].Q THEN
	stAlarm.arrFlowAlarm[39]:=TRUE;//NG料盒料满报警
END_IF

///NG踢废堵料报警
IF tonAuto[31].Q THEN
	stAlarm.arrFlowAlarm[44]:=TRUE;//NG踢废堵料报警
END_IF

//分段皮带3料盒满料报警
IF (iPartSelect=1 AND tonAuto[28].Q) OR (iPartSelect=2 AND  tonAuto[29].Q) THEN
	stAlarm.arrFlowAlarm[43]:=TRUE;//分段皮带3料盒满料报警
END_IF

//单位时间内NG个数
IF NOT tonAuto[22].Q THEN
	tonAuto[22].IN:=TRUE;
ELSE
	IF NG_Sum>=ProductPar.iModeEN.iNGPole THEN
		stAlarm.arrFlowAlarm[26]:=TRUE;
	END_IF
	NG_Sum:=0;
	tonAuto[22].IN:=FALSE;
END_IF
IF arrCyCtrl[CYNo.NGRevBeltUpDown].Cmd.bOFF THEN
	stAlarm.arrLightWarn[23]:=TRUE;
END_IF


